LIN {X 0,Y 514.336,Z 499.289,A -85,B 0,C 180,E1 19058.473,E2 19058.473} C_VEL
LIN {X 0,Y 521.666,Z 511.936,A -85,B 0,C 180,E1 19056.114,E2 19056.114} C_VEL
LIN {X 0,Y 522.287,Z 513.297,A -85,B 0,C 180,E1 19055.918,E2 19055.918} C_VEL
LIN {X 0,Y 507.153,Z 734.617,A -85,B 0,C 180,E1 19052.471,E2 19052.471} C_VEL
LIN {X 0,Y 501.246,Z 821.128,A -85,B 0,C 180,E1 19051.105,E2 19051.105} C_VEL
LIN {X 0,Y 497.966,Z 849.233,A -85,B 0,C 180,E1 19050.568,E2 19050.568} C_VEL
LIN {X 0,Y 493.711,Z 874.723,A -85,B 0,C 180,E1 19049.927,E2 19049.927} C_VEL
LIN {X 0,Y 489.478,Z 895.998,A -85,B 0,C 180,E1 19049.256,E2 19049.256} C_VEL
LIN {X 0,Y 484.89,Z 916.021,A -85,B 0,C 180,E1 19048.501,E2 19048.501} C_VEL
LIN {X 0,Y 479.636,Z 936.391,A -85,B 0,C 180,E1 19047.593,E2 19047.593} C_VEL
LIN {X 0,Y 472.466,Z 961.41,A -85,B 0,C 180,E1 19046.272,E2 19046.272} C_VEL
LIN {X 0,Y 464.663,Z 985.247,A -85,B 0,C 180,E1 19044.746,E2 19044.746} C_VEL
LIN {X 0,Y 457.779,Z 1004.83,A -85,B 0,C 180,E1 19043.281,E2 19043.281} C_VEL
LIN {X 0,Y 450.93,Z 1023.119,A -85,B 0,C 180,E1 19041.714,E2 19041.714} C_VEL
LIN {X 0,Y 442.952,Z 1043.356,A -85,B 0,C 180,E1 19039.725,E2 19039.725} C_VEL
LIN {X 0,Y 434.117,Z 1064.457,A -85,B 0,C 180,E1 19037.283,E2 19037.283} C_VEL
LIN {X 0,Y 427.056,Z 1080.83,A -85,B 0,C 180,E1 19035.092,E2 19035.092} C_VEL
LIN {X 0,Y 420.572,Z 1095.666,A -85,B 0,C 180,E1 19032.838,E2 19032.838} C_VEL
LIN {X 0,Y 414.005,Z 1110.651,A -85,B 0,C 180,E1 19030.253,E2 19030.253} C_VEL
LIN {X 0,Y 406.387,Z 1128.256,A -85,B 0,C 180,E1 19026.717,E2 19026.717} C_VEL
LIN {X 0,Y 400.867,Z 1141.384,A -85,B 0,C 180,E1 19023.623,E2 19023.623} C_VEL
LIN {X 0,Y 396.527,Z 1152.254,A -85,B 0,C 180,E1 19020.697,E2 19020.697} C_VEL
LIN {X 0,Y 392.827,Z 1162.333,A -85,B 0,C 180,E1 19017.596,E2 19017.596} C_VEL
LIN {X 0,Y 389.21,Z 1173.396,A -85,B 0,C 180,E1 19013.625,E2 19013.625} C_VEL
LIN {X 0,Y 386.872,Z 1181.783,A -85,B 0,C 180,E1 19009.947,E2 19009.947} C_VEL
LIN {X 0,Y 385.478,Z 1187.928,A -85,B 0,C 180,E1 19006.733,E2 19006.733} C_VEL
LIN {X 0,Y 384.662,Z 1192.751,A -85,B 0,C 180,E1 19003.682,E2 19003.682} C_VEL
LIN {X 0,Y 384.204,Z 1196.587,A -85,B 0,C 180,E1 19000.648,E2 19000.648} C_VEL
LIN {X 0,Y 384.01,Z 1199.46,A -85,B 0,C 180,E1 18997.631,E2 18997.631} C_VEL
LIN {X 0,Y 383.947,Z 1201.384,A -85,B 0,C 180,E1 18994.63,E2 18994.63} C_VEL
LIN {X 0,Y 383.945,Z 1202.344,A -85,B 0,C 180,E1 18991.791,E2 18991.791} C_VEL
LIN {X 0,Y 383.945,Z 1202.461,A -85,B 0,C 180,E1 18988.955,E2 18988.955} C_VEL
LIN {X 0,Y 383.943,Z 1201.632,A -85,B 0,C 180,E1 18985.899,E2 18985.899} C_VEL
LIN {X 0,Y 383.992,Z 1199.811,A -85,B 0,C 180,E1 18982.82,E2 18982.82} C_VEL
LIN {X 0,Y 384.164,Z 1197.081,A -85,B 0,C 180,E1 18979.806,E2 18979.806} C_VEL
LIN {X 0,Y 384.565,Z 1193.388,A -85,B 0,C 180,E1 18976.774,E2 18976.774} C_VEL
LIN {X 0,Y 385.339,Z 1188.712,A -85,B 0,C 180,E1 18973.726,E2 18973.726} C_VEL
LIN {X 0,Y 386.553,Z 1183.024,A -85,B 0,C 180,E1 18970.665,E2 18970.665} C_VEL
LIN {X 0,Y 388.357,Z 1176.207,A -85,B 0,C 180,E1 18967.565,E2 18967.565} C_VEL
LIN {X 0,Y 390.867,Z 1168.055,A -85,B 0,C 180,E1 18964.386,E2 18964.386} C_VEL
LIN {X 0,Y 394.947,Z 1156.625,A -85,B 0,C 180,E1 18960.565,E2 18960.565} C_VEL
LIN {X 0,Y 399.901,Z 1143.712,A -85,B 0,C 180,E1 18956.972,E2 18956.972} C_VEL
LIN {X 0,Y 404.792,Z 1131.925,A -85,B 0,C 180,E1 18954.116,E2 18954.116} C_VEL
LIN {X 0,Y 410.265,Z 1119.184,A -85,B 0,C 180,E1 18951.399,E2 18951.399} C_VEL
LIN {X 0,Y 416.577,Z 1104.778,A -85,B 0,C 180,E1 18948.697,E2 18948.697} C_VEL
LIN {X 0,Y 425.211,Z 1085.008,A -85,B 0,C 180,E1 18945.515,E2 18945.515} C_VEL
LIN {X 0,Y 432.324,Z 1068.503,A -85,B 0,C 180,E1 18943.238,E2 18943.238} C_VEL
LIN {X 0,Y 439.276,Z 1052.004,A -85,B 0,C 180,E1 18941.239,E2 18941.239} C_VEL
LIN {X 0,Y 446.663,Z 1033.856,A -85,B 0,C 180,E1 18939.31,E2 18939.31} C_VEL
LIN {X 0,Y 455.882,Z 1009.897,A -85,B 0,C 180,E1 18937.133,E2 18937.133} C_VEL
LIN {X 0,Y 463.244,Z 989.199,A -85,B 0,C 180,E1 18935.54,E2 18935.54} C_VEL
LIN {X 0,Y 469.526,Z 970.341,A -85,B 0,C 180,E1 18934.285,E2 18934.285} C_VEL
LIN {X 0,Y 475.391,Z 951.136,A -85,B 0,C 180,E1 18933.167,E2 18933.167} C_VEL
LIN {X 0,Y 481.322,Z 929.886,A -85,B 0,C 180,E1 18932.106,E2 18932.106} C_VEL
LIN {X 0,Y 488.036,Z 902.402,A -85,B 0,C 180,E1 18930.975,E2 18930.975} C_VEL
LIN {X 0,Y 492.871,Z 878.77,A -85,B 0,C 180,E1 18930.196,E2 18930.196} C_VEL
LIN {X 0,Y 496.583,Z 857.355,A -85,B 0,C 180,E1 18929.628,E2 18929.628} C_VEL
LIN {X 0,Y 499.707,Z 834.953,A -85,B 0,C 180,E1 18929.153,E2 18929.153} C_VEL
LIN {X 0,Y 502.37,Z 806.226,A -85,B 0,C 180,E1 18928.651,E2 18928.651} C_VEL
LIN {X 0,Y 517.218,Z 584.32,A -85,B 0,C 180,E1 18925.194,E2 18925.194} C_VEL
LIN {X 0,Y 522.155,Z 512.95,A -85,B 0,C 180,E1 18924.072,E2 18924.072} C_VEL
LIN {X 0,Y 515.699,Z 501.805,A -85,B 0,C 180,E1 18922.035,E2 18922.035} C_VEL
LIN {X 0,Y 508.977,Z 490.578,A -85,B 0,C 180,E1 18919.659,E2 18919.659} C_VEL
LIN {X 0,Y 502.568,Z 480.516,A -85,B 0,C 180,E1 18917.065,E2 18917.065} C_VEL
LIN {X 0,Y 498.85,Z 474.804,A -85,B 0,C 180,E1 18915.342,E2 18915.342} C_VEL
LIN {X 0,Y 494.845,Z 469.392,A -85,B 0,C 180,E1 18913.258,E2 18913.258} C_VEL
LIN {X 0,Y 491.244,Z 464.512,A -85,B 0,C 180,E1 18911.03,E2 18911.03} C_VEL
LIN {X 0,Y 488.198,Z 460.623,A -85,B 0,C 180,E1 18908.717,E2 18908.717} C_VEL
LIN {X 0,Y 487.346,Z 459.062,A -85,B 0,C 180,E1 18907.901,E2 18907.901} C_VEL
LIN {X 0,Y 484.26,Z 455.669,A -85,B 0,C 180,E1 18904.144,E2 18904.144} C_VEL
LIN {X 0,Y 483.557,Z 453.202,A -85,B 0,C 180,E1 18902.133,E2 18902.133} C_VEL
LIN {X 0,Y 483.631,Z 453.363,A -85,B 0,C 180,E1 18897.109,E2 18897.109} C_VEL
LIN {X 0,Y 485.036,Z 457.019,A -85,B 0,C 180,E1 18894.084,E2 18894.084} C_VEL
LIN {X 0,Y 487.613,Z 459.507,A -85,B 0,C 180,E1 18891.331,E2 18891.331} C_VEL
LIN {X 0,Y 490.183,Z 463.479,A -85,B 0,C 180,E1 18889.183,E2 18889.183} C_VEL
LIN {X 0,Y 491.887,Z 465.368,A -85,B 0,C 180,E1 18888.033,E2 18888.033} C_VEL
LIN {X 0,Y 495.311,Z 469.926,A -85,B 0,C 180,E1 18885.981,E2 18885.981} C_VEL
LIN {X 0,Y 500.203,Z 476.705,A -85,B 0,C 180,E1 18883.51,E2 18883.51} C_VEL
LIN {X 0,Y 504.513,Z 482.766,A -85,B 0,C 180,E1 18881.632,E2 18881.632} C_VEL
LIN {X 0,Y 509.943,Z 490.429,A -85,B 0,C 180,E1 18879.543,E2 18879.543} C_VEL
LIN {X 0,Y 518.713,Z 503.424,A -85,B 0,C 180,E1 18876.603,E2 18876.603} C_VEL
LIN {X 0,Y 522.118,Z 509.067,A -85,B 0,C 180,E1 18875.558,E2 18875.558} C_VEL
LIN {X 0,Y 507.325,Z 724.277,A -85,B 0,C 180,E1 18872.21,E2 18872.21} C_VEL
LIN {X 0,Y 501.73,Z 805.31,A -85,B 0,C 180,E1 18870.931,E2 18870.931} C_VEL
LIN {X 0,Y 498.508,Z 833.243,A -85,B 0,C 180,E1 18870.382,E2 18870.382} C_VEL
LIN {X 0,Y 494.471,Z 858.277,A -85,B 0,C 180,E1 18869.718,E2 18869.718} C_VEL
LIN {X 0,Y 490.363,Z 879.378,A -85,B 0,C 180,E1 18869.026,E2 18869.026} C_VEL
LIN {X 0,Y 485.757,Z 899.843,A -85,B 0,C 180,E1 18868.222,E2 18868.222} C_VEL
LIN {X 0,Y 480.065,Z 922.038,A -85,B 0,C 180,E1 18867.192,E2 18867.192} C_VEL
LIN {X 0,Y 472.51,Z 947.879,A -85,B 0,C 180,E1 18865.744,E2 18865.744} C_VEL
LIN {X 0,Y 465.938,Z 967.878,A -85,B 0,C 180,E1 18864.419,E2 18864.419} C_VEL
LIN {X 0,Y 459.376,Z 986.337,A -85,B 0,C 180,E1 18863.015,E2 18863.015} C_VEL
LIN {X 0,Y 452.562,Z 1004.295,A -85,B 0,C 180,E1 18861.453,E2 18861.453} C_VEL
LIN {X 0,Y 444.578,Z 1024.231,A -85,B 0,C 180,E1 18859.459,E2 18859.459} C_VEL
LIN {X 0,Y 435.572,Z 1045.248,A -85,B 0,C 180,E1 18856.98,E2 18856.98} C_VEL
LIN {X 0,Y 428.495,Z 1061.153,A -85,B 0,C 180,E1 18854.805,E2 18854.805} C_VEL
LIN {X 0,Y 421.79,Z 1075.935,A -85,B 0,C 180,E1 18852.5,E2 18852.5} C_VEL
LIN {X 0,Y 414.34,Z 1092.31,A -85,B 0,C 180,E1 18849.573,E2 18849.573} C_VEL
LIN {X 0,Y 407.177,Z 1107.877,A -85,B 0,C 180,E1 18846.284,E2 18846.284} C_VEL
LIN {X 0,Y 401.812,Z 1119.823,A -85,B 0,C 180,E1 18843.362,E2 18843.362} C_VEL
LIN {X 0,Y 397.504,Z 1129.916,A -85,B 0,C 180,E1 18840.537,E2 18840.537} C_VEL
LIN {X 0,Y 393.556,Z 1139.762,A -85,B 0,C 180,E1 18837.377,E2 18837.377} C_VEL
LIN {X 0,Y 389.661,Z 1150.554,A -85,B 0,C 180,E1 18833.27,E2 18833.27} C_VEL
LIN {X 0,Y 387.29,Z 1158.095,A -85,B 0,C 180,E1 18829.767,E2 18829.767} C_VEL
LIN {X 0,Y 385.802,Z 1163.853,A -85,B 0,C 180,E1 18826.564,E2 18826.564} C_VEL
LIN {X 0,Y 384.832,Z 1168.546,A -85,B 0,C 180,E1 18823.37,E2 18823.37} C_VEL
LIN {X 0,Y 384.304,Z 1172.209,A -85,B 0,C 180,E1 18820.19,E2 18820.19} C_VEL
LIN {X 0,Y 384.054,Z 1174.876,A -85,B 0,C 180,E1 18817.028,E2 18817.028} C_VEL
LIN {X 0,Y 383.964,Z 1176.634,A -85,B 0,C 180,E1 18813.733,E2 18813.733} C_VEL
LIN {X 0,Y 383.95,Z 1177.409,A -85,B 0,C 180,E1 18810,E2 18810} C_VEL
LIN {X 0,Y 383.964,Z 1176.675,A -85,B 0,C 180,E1 18806.267,E2 18806.267} C_VEL
LIN {X 0,Y 384.048,Z 1174.945,A -85,B 0,C 180,E1 18802.972,E2 18802.972} C_VEL
LIN {X 0,Y 384.075,Z 1174.587,A -85,B 0,C 180,E1 18802.483,E2 18802.483} C_VEL
LIN {X 0,Y 383.137,Z 1173.813,A -85,B 0,C 180,E1 18801.338,E2 18801.338} C_VEL
LIN {X 0,Y 377.082,Z 1171.119,A -85,B 0,C 180,E1 18798.109,E2 18798.109} C_VEL
LIN {X 0,Y 376.701,Z 1170.137,A -85,B 0,C 180,E1 18797.275,E2 18797.275} C_VEL
LIN {X 0,Y 377.746,Z 1165.009,A -85,B 0,C 180,E1 18793.548,E2 18793.548} C_VEL
LIN {X 0,Y 379.241,Z 1159.399,A -85,B 0,C 180,E1 18790.263,E2 18790.263} C_VEL
LIN {X 0,Y 381.436,Z 1152.594,A -85,B 0,C 180,E1 18786.942,E2 18786.942} C_VEL
LIN {X 0,Y 384.593,Z 1144.069,A -85,B 0,C 180,E1 18783.426,E2 18783.426} C_VEL
LIN {X 0,Y 389.595,Z 1131.982,A -85,B 0,C 180,E1 18779.289,E2 18779.289} C_VEL
LIN {X 0,Y 394.485,Z 1120.971,A -85,B 0,C 180,E1 18776.109,E2 18776.109} C_VEL
LIN {X 0,Y 399.733,Z 1109.743,A -85,B 0,C 180,E1 18773.287,E2 18773.287} C_VEL
LIN {X 0,Y 405.907,Z 1096.826,A -85,B 0,C 180,E1 18770.447,E2 18770.447} C_VEL
LIN {X 0,Y 414.365,Z 1079.157,A -85,B 0,C 180,E1 18767.12,E2 18767.12} C_VEL
LIN {X 0,Y 422.034,Z 1062.829,A -85,B 0,C 180,E1 18764.512,E2 18764.512} C_VEL
LIN {X 0,Y 429.08,Z 1047.553,A -85,B 0,C 180,E1 18762.381,E2 18762.381} C_VEL
LIN {X 0,Y 436.644,Z 1030.627,A -85,B 0,C 180,E1 18760.313,E2 18760.313} C_VEL
LIN {X 0,Y 446.241,Z 1007.9,A -85,B 0,C 180,E1 18757.936,E2 18757.936} C_VEL
LIN {X 0,Y 453.74,Z 988.819,A -85,B 0,C 180,E1 18756.244,E2 18756.244} C_VEL
LIN {X 0,Y 460.515,Z 970.415,A -85,B 0,C 180,E1 18754.823,E2 18754.823} C_VEL
LIN {X 0,Y 466.515,Z 952.797,A -85,B 0,C 180,E1 18753.628,E2 18753.628} C_VEL
LIN {X 0,Y 472.745,Z 932.837,A -85,B 0,C 180,E1 18752.447,E2 18752.447} C_VEL
LIN {X 0,Y 479.8,Z 907.755,A -85,B 0,C 180,E1 18751.192,E2 18751.192} C_VEL
LIN {X 0,Y 485.738,Z 882.561,A -85,B 0,C 180,E1 18750.17,E2 18750.17} C_VEL
LIN {X 0,Y 490.062,Z 861.218,A -85,B 0,C 180,E1 18749.456,E2 18749.456} C_VEL
LIN {X 0,Y 493.656,Z 840.065,A -85,B 0,C 180,E1 18748.875,E2 18748.875} C_VEL
LIN {X 0,Y 496.845,Z 816.624,A -85,B 0,C 180,E1 18748.365,E2 18748.365} C_VEL
LIN {X 0,Y 499.925,Z 780.742,A -85,B 0,C 180,E1 18747.765,E2 18747.765} C_VEL
LIN {X 0,Y 515.453,Z 558.007,A -85,B 0,C 180,E1 18744.299,E2 18744.299} C_VEL
LIN {X 0,Y 518.584,Z 513.689,A -85,B 0,C 180,E1 18743.59,E2 18743.59} C_VEL
LIN {X 0,Y 510.496,Z 501.292,A -85,B 0,C 180,E1 18740.914,E2 18740.914} C_VEL
LIN {X 0,Y 503.874,Z 491.617,A -85,B 0,C 180,E1 18738.392,E2 18738.392} C_VEL
LIN {X 0,Y 499.546,Z 485.536,A -85,B 0,C 180,E1 18736.513,E2 18736.513} C_VEL
LIN {X 0,Y 496.88,Z 481.827,A -85,B 0,C 180,E1 18735.225,E2 18735.225} C_VEL
LIN {X 0,Y 493.53,Z 477.194,A -85,B 0,C 180,E1 18733.414,E2 18733.414} C_VEL
LIN {X 0,Y 490.037,Z 472.267,A -85,B 0,C 180,E1 18731.177,E2 18731.177} C_VEL
LIN {X 0,Y 487.021,Z 468.411,A -85,B 0,C 180,E1 18728.798,E2 18728.798} C_VEL
LIN {X 0,Y 486.273,Z 466.929,A -85,B 0,C 180,E1 18728.038,E2 18728.038} C_VEL
LIN {X 0,Y 483.192,Z 463.339,A -85,B 0,C 180,E1 18723.916,E2 18723.916} C_VEL
LIN {X 0,Y 482.689,Z 461.161,A -85,B 0,C 180,E1 18722.018,E2 18722.018} C_VEL
LIN {X 0,Y 482.758,Z 461.298,A -85,B 0,C 180,E1 18718.101,E2 18718.101} C_VEL
LIN {X 0,Y 484.664,Z 465.68,A -85,B 0,C 180,E1 18714.079,E2 18714.079} C_VEL
LIN {X 0,Y 486.62,Z 467.409,A -85,B 0,C 180,E1 18712.038,E2 18712.038} C_VEL
LIN {X 0,Y 489.444,Z 471.765,A -85,B 0,C 180,E1 18709.643,E2 18709.643} C_VEL
LIN {X 0,Y 490.79,Z 473.291,A -85,B 0,C 180,E1 18708.721,E2 18708.721} C_VEL
LIN {X 0,Y 494.745,Z 478.782,A -85,B 0,C 180,E1 18706.322,E2 18706.322} C_VEL
LIN {X 0,Y 498.948,Z 484.683,A -85,B 0,C 180,E1 18704.184,E2 18704.184} C_VEL
LIN {X 0,Y 505.315,Z 494.859,A -85,B 0,C 180,E1 18701.393,E2 18701.393} C_VEL
LIN {X 0,Y 512.231,Z 506.445,A -85,B 0,C 180,E1 18698.801,E2 18698.801} C_VEL
LIN {X 0,Y 518.7,Z 517.874,A -85,B 0,C 180,E1 18696.655,E2 18696.655} C_VEL
LIN {X 0,Y 503.228,Z 738.076,A -85,B 0,C 180,E1 18693.226,E2 18693.226} C_VEL
LIN {X 0,Y 497.396,Z 820.991,A -85,B 0,C 180,E1 18691.915,E2 18691.915} C_VEL
LIN {X 0,Y 494.008,Z 849.281,A -85,B 0,C 180,E1 18691.374,E2 18691.374} C_VEL
LIN {X 0,Y 489.714,Z 874.468,A -85,B 0,C 180,E1 18690.744,E2 18690.744} C_VEL
LIN {X 0,Y 485.383,Z 895.74,A -85,B 0,C 180,E1 18690.079,E2 18690.079} C_VEL
LIN {X 0,Y 480.691,Z 915.761,A -85,B 0,C 180,E1 18689.327,E2 18689.327} C_VEL
LIN {X 0,Y 475.177,Z 936.612,A -85,B 0,C 180,E1 18688.402,E2 18688.402} C_VEL
LIN {X 0,Y 467.654,Z 962.063,A -85,B 0,C 180,E1 18687.053,E2 18687.053} C_VEL
LIN {X 0,Y 459.937,Z 985.028,A -85,B 0,C 180,E1 18685.581,E2 18685.581} C_VEL
LIN {X 0,Y 453.16,Z 1003.821,A -85,B 0,C 180,E1 18684.179,E2 18684.179} C_VEL
LIN {X 0,Y 446.355,Z 1021.501,A -85,B 0,C 180,E1 18682.676,E2 18682.676} C_VEL
LIN {X 0,Y 439.084,Z 1039.394,A -85,B 0,C 180,E1 18680.942,E2 18680.942} C_VEL
LIN {X 0,Y 430.172,Z 1060.455,A -85,B 0,C 180,E1 18678.581,E2 18678.581} C_VEL
LIN {X 0,Y 421.59,Z 1079.621,A -85,B 0,C 180,E1 18676.037,E2 18676.037} C_VEL
LIN {X 0,Y 414.823,Z 1094.533,A -85,B 0,C 180,E1 18673.77,E2 18673.77} C_VEL
LIN {X 0,Y 408.469,Z 1108.461,A -85,B 0,C 180,E1 18671.369,E2 18671.369} C_VEL
LIN {X 0,Y 402.092,Z 1122.506,A -85,B 0,C 180,E1 18668.619,E2 18668.619} C_VEL
LIN {X 0,Y 394.623,Z 1139.351,A -85,B 0,C 180,E1 18664.756,E2 18664.756} C_VEL
LIN {X 0,Y 389.639,Z 1151.167,A -85,B 0,C 180,E1 18661.566,E2 18661.566} C_VEL
LIN {X 0,Y 385.737,Z 1161.118,A -85,B 0,C 180,E1 18658.486,E2 18658.486} C_VEL
LIN {X 0,Y 382.35,Z 1170.7,A -85,B 0,C 180,E1 18655.064,E2 18655.064} C_VEL
LIN {X 0,Y 379.258,Z 1180.887,A -85,B 0,C 180,E1 18650.687,E2 18650.687} C_VEL
LIN {X 0,Y 377.652,Z 1187.396,A -85,B 0,C 180,E1 18647.249,E2 18647.249} C_VEL
LIN {X 0,Y 376.724,Z 1192.483,A -85,B 0,C 180,E1 18643.976,E2 18643.976} C_VEL
LIN {X 0,Y 376.224,Z 1196.321,A -85,B 0,C 180,E1 18640.876,E2 18640.876} C_VEL
LIN {X 0,Y 376.015,Z 1199.196,A -85,B 0,C 180,E1 18637.794,E2 18637.794} C_VEL
LIN {X 0,Y 375.953,Z 1201.05,A -85,B 0,C 180,E1 18634.882,E2 18634.882} C_VEL
LIN {X 0,Y 375.949,Z 1202.081,A -85,B 0,C 180,E1 18631.829,E2 18631.829} C_VEL
LIN {X 0,Y 375.95,Z 1202.198,A -85,B 0,C 180,E1 18628.933,E2 18628.933} C_VEL
LIN {X 0,Y 375.946,Z 1201.387,A -85,B 0,C 180,E1 18625.851,E2 18625.851} C_VEL
LIN {X 0,Y 376.005,Z 1199.547,A -85,B 0,C 180,E1 18622.667,E2 18622.667} C_VEL
LIN {X 0,Y 376.184,Z 1196.789,A -85,B 0,C 180,E1 18619.564,E2 18619.564} C_VEL
LIN {X 0,Y 376.654,Z 1192.906,A -85,B 0,C 180,E1 18616.334,E2 18616.334} C_VEL
LIN {X 0,Y 377.487,Z 1188.179,A -85,B 0,C 180,E1 18613.219,E2 18613.219} C_VEL
LIN {X 0,Y 378.906,Z 1182.17,A -85,B 0,C 180,E1 18609.959,E2 18609.959} C_VEL
LIN {X 0,Y 381.081,Z 1174.564,A -85,B 0,C 180,E1 18606.496,E2 18606.496} C_VEL
LIN {X 0,Y 384.895,Z 1163.457,A -85,B 0,C 180,E1 18602.29,E2 18602.29} C_VEL
LIN {X 0,Y 389.044,Z 1152.603,A -85,B 0,C 180,E1 18598.854,E2 18598.854} C_VEL
LIN {X 0,Y 393.608,Z 1141.677,A -85,B 0,C 180,E1 18595.848,E2 18595.848} C_VEL
LIN {X 0,Y 399.04,Z 1129.249,A -85,B 0,C 180,E1 18592.853,E2 18592.853} C_VEL
LIN {X 0,Y 406.354,Z 1113.12,A -85,B 0,C 180,E1 18589.49,E2 18589.49} C_VEL
LIN {X 0,Y 413.642,Z 1097.059,A -85,B 0,C 180,E1 18586.647,E2 18586.647} C_VEL
LIN {X 0,Y 420.509,Z 1081.911,A -85,B 0,C 180,E1 18584.3,E2 18584.3} C_VEL
LIN {X 0,Y 427.535,Z 1066.17,A -85,B 0,C 180,E1 18582.153,E2 18582.153} C_VEL
LIN {X 0,Y 435.234,Z 1048.451,A -85,B 0,C 180,E1 18580.036,E2 18580.036} C_VEL
LIN {X 0,Y 444.756,Z 1025.434,A -85,B 0,C 180,E1 18577.69,E2 18577.69} C_VEL
LIN {X 0,Y 452.304,Z 1005.911,A -85,B 0,C 180,E1 18575.995,E2 18575.995} C_VEL
LIN {X 0,Y 459.066,Z 987.286,A -85,B 0,C 180,E1 18574.584,E2 18574.584} C_VEL
LIN {X 0,Y 465.827,Z 967.344,A -85,B 0,C 180,E1 18573.277,E2 18573.277} C_VEL
LIN {X 0,Y 473.448,Z 942.736,A -85,B 0,C 180,E1 18571.901,E2 18571.901} C_VEL
LIN {X 0,Y 480.033,Z 918.088,A -85,B 0,C 180,E1 18570.774,E2 18570.774} C_VEL
LIN {X 0,Y 485.038,Z 896.924,A -85,B 0,C 180,E1 18569.968,E2 18569.968} C_VEL
LIN {X 0,Y 489.485,Z 875.199,A -85,B 0,C 180,E1 18569.282,E2 18569.282} C_VEL
LIN {X 0,Y 493.495,Z 851.865,A -85,B 0,C 180,E1 18568.692,E2 18568.692} C_VEL
LIN {X 0,Y 497.217,Z 821.963,A -85,B 0,C 180,E1 18568.108,E2 18568.108} C_VEL
LIN {X 0,Y 501.928,Z 755.768,A -85,B 0,C 180,E1 18567.056,E2 18567.056} C_VEL
LIN {X 0,Y 517.35,Z 534.967,A -85,B 0,C 180,E1 18563.617,E2 18563.617} C_VEL
LIN {X 0,Y 518.578,Z 517.678,A -85,B 0,C 180,E1 18563.343,E2 18563.343} C_VEL
LIN {X 0,Y 511.57,Z 505.471,A -85,B 0,C 180,E1 18561.018,E2 18561.018} C_VEL
LIN {X 0,Y 504.833,Z 494.213,A -85,B 0,C 180,E1 18558.476,E2 18558.476} C_VEL
LIN {X 0,Y 498.44,Z 484.005,A -85,B 0,C 180,E1 18555.653,E2 18555.653} C_VEL
LIN {X 0,Y 493.462,Z 477.084,A -85,B 0,C 180,E1 18553.058,E2 18553.058} C_VEL
LIN {X 0,Y 489.925,Z 472.243,A -85,B 0,C 180,E1 18550.822,E2 18550.822} C_VEL
LIN {X 0,Y 486.957,Z 468.311,A -85,B 0,C 180,E1 18548.502,E2 18548.502} C_VEL
LIN {X 0,Y 486.245,Z 466.949,A -85,B 0,C 180,E1 18547.8,E2 18547.8} C_VEL
LIN {X 0,Y 483.22,Z 463.549,A -85,B 0,C 180,E1 18544.034,E2 18544.034} C_VEL
LIN {X 0,Y 482.543,Z 461.136,A -85,B 0,C 180,E1 18542.019,E2 18542.019} C_VEL
LIN {X 0,Y 482.631,Z 461.368,A -85,B 0,C 180,E1 18537.15,E2 18537.15} C_VEL
LIN {X 0,Y 484.145,Z 465.133,A -85,B 0,C 180,E1 18533.954,E2 18533.954} C_VEL
LIN {X 0,Y 486.446,Z 467.331,A -85,B 0,C 180,E1 18531.489,E2 18531.489} C_VEL
LIN {X 0,Y 489.049,Z 471.365,A -85,B 0,C 180,E1 18529.277,E2 18529.277} C_VEL
LIN {X 0,Y 490.559,Z 473.066,A -85,B 0,C 180,E1 18528.239,E2 18528.239} C_VEL
LIN {X 0,Y 494.723,Z 478.899,A -85,B 0,C 180,E1 18525.725,E2 18525.725} C_VEL
LIN {X 0,Y 498.62,Z 484.252,A -85,B 0,C 180,E1 18523.755,E2 18523.755} C_VEL
LIN {X 0,Y 502.729,Z 490.13,A -85,B 0,C 180,E1 18521.924,E2 18521.924} C_VEL
LIN {X 0,Y 508.137,Z 497.92,A -85,B 0,C 180,E1 18519.797,E2 18519.797} C_VEL
LIN {X 0,Y 516.54,Z 510.577,A -85,B 0,C 180,E1 18516.922,E2 18516.922} C_VEL
LIN {X 0,Y 518.519,Z 513.964,A -85,B 0,C 180,E1 18516.292,E2 18516.292} C_VEL
LIN {X 0,Y 503.283,Z 729.841,A -85,B 0,C 180,E1 18512.933,E2 18512.933} C_VEL
LIN {X 0,Y 497.871,Z 805.809,A -85,B 0,C 180,E1 18511.733,E2 18511.733} C_VEL
LIN {X 0,Y 494.513,Z 834.039,A -85,B 0,C 180,E1 18511.177,E2 18511.177} C_VEL
LIN {X 0,Y 490.451,Z 858.66,A -85,B 0,C 180,E1 18510.524,E2 18510.524} C_VEL
LIN {X 0,Y 486.27,Z 879.653,A -85,B 0,C 180,E1 18509.839,E2 18509.839} C_VEL
LIN {X 0,Y 481.556,Z 900.117,A -85,B 0,C 180,E1 18509.038,E2 18509.038} C_VEL
LIN {X 0,Y 475.787,Z 922.096,A -85,B 0,C 180,E1 18508.022,E2 18508.022} C_VEL
LIN {X 0,Y 467.931,Z 948.312,A -85,B 0,C 180,E1 18506.556,E2 18506.556} C_VEL
LIN {X 0,Y 461.202,Z 968.25,A -85,B 0,C 180,E1 18505.237,E2 18505.237} C_VEL
LIN {X 0,Y 454.498,Z 986.61,A -85,B 0,C 180,E1 18503.839,E2 18503.839} C_VEL
LIN {X 0,Y 447.495,Z 1004.569,A -85,B 0,C 180,E1 18502.275,E2 18502.275} C_VEL
LIN {X 0,Y 439.564,Z 1023.79,A -85,B 0,C 180,E1 18500.351,E2 18500.351} C_VEL
LIN {X 0,Y 430.196,Z 1045.024,A -85,B 0,C 180,E1 18497.852,E2 18497.852} C_VEL
LIN {X 0,Y 422.645,Z 1061.428,A -85,B 0,C 180,E1 18495.598,E2 18495.598} C_VEL
LIN {X 0,Y 415.693,Z 1076.211,A -85,B 0,C 180,E1 18493.275,E2 18493.275} C_VEL
LIN {X 0,Y 407.942,Z 1092.586,A -85,B 0,C 180,E1 18490.32,E2 18490.32} C_VEL
LIN {X 0,Y 400.416,Z 1108.295,A -85,B 0,C 180,E1 18486.957,E2 18486.957} C_VEL
LIN {X 0,Y 394.877,Z 1120.099,A -85,B 0,C 180,E1 18484.027,E2 18484.027} C_VEL
LIN {X 0,Y 390.341,Z 1130.192,A -85,B 0,C 180,E1 18481.159,E2 18481.159} C_VEL
LIN {X 0,Y 386.188,Z 1140.037,A -85,B 0,C 180,E1 18477.944,E2 18477.944} C_VEL
LIN {X 0,Y 382.07,Z 1150.816,A -85,B 0,C 180,E1 18473.766,E2 18473.766} C_VEL
LIN {X 0,Y 379.545,Z 1158.367,A -85,B 0,C 180,E1 18470.188,E2 18470.188} C_VEL
LIN {X 0,Y 377.949,Z 1164.123,A -85,B 0,C 180,E1 18466.918,E2 18466.918} C_VEL
LIN {X 0,Y 376.92,Z 1168.814,A -85,B 0,C 180,E1 18463.656,E2 18463.656} C_VEL
LIN {X 0,Y 376.342,Z 1172.475,A -85,B 0,C 180,E1 18460.408,E2 18460.408} C_VEL
LIN {X 0,Y 376.072,Z 1175.14,A -85,B 0,C 180,E1 18457.178,E2 18457.178} C_VEL
LIN {X 0,Y 375.97,Z 1176.897,A -85,B 0,C 180,E1 18453.812,E2 18453.812} C_VEL
LIN {X 0,Y 375.954,Z 1177.672,A -85,B 0,C 180,E1 18450,E2 18450} C_VEL
LIN {X 0,Y 375.97,Z 1176.938,A -85,B 0,C 180,E1 18446.188,E2 18446.188} C_VEL
LIN {X 0,Y 376.064,Z 1175.208,A -85,B 0,C 180,E1 18442.822,E2 18442.822} C_VEL
LIN {X 0,Y 376.331,Z 1172.57,A -85,B 0,C 180,E1 18439.591,E2 18439.591} C_VEL
LIN {X 0,Y 376.701,Z 1170.137,A -85,B 0,C 180,E1 18437.275,E2 18437.275} C_VEL
LIN {X 0,Y 375.953,Z 1168.761,A -85,B 0,C 180,E1 18436.12,E2 18436.12} C_VEL
LIN {X 0,Y 370.608,Z 1164.818,A -85,B 0,C 180,E1 18432.924,E2 18432.924} C_VEL
LIN {X 0,Y 370.384,Z 1163.436,A -85,B 0,C 180,E1 18431.999,E2 18431.999} C_VEL
LIN {X 0,Y 373.048,Z 1155.068,A -85,B 0,C 180,E1 18427.463,E2 18427.463} C_VEL
LIN {X 0,Y 376.016,Z 1147.133,A -85,B 0,C 180,E1 18423.976,E2 18423.976} C_VEL
LIN {X 0,Y 379.513,Z 1138.773,A -85,B 0,C 180,E1 18420.83,E2 18420.83} C_VEL
LIN {X 0,Y 383.817,Z 1129.234,A -85,B 0,C 180,E1 18417.722,E2 18417.722} C_VEL
LIN {X 0,Y 389.813,Z 1116.753,A -85,B 0,C 180,E1 18414.21,E2 18414.21} C_VEL
LIN {X 0,Y 397.256,Z 1101.581,A -85,B 0,C 180,E1 18410.635,E2 18410.635} C_VEL
LIN {X 0,Y 403.782,Z 1088.477,A -85,B 0,C 180,E1 18407.979,E2 18407.979} C_VEL
LIN {X 0,Y 410.663,Z 1074.59,A -85,B 0,C 180,E1 18405.513,E2 18405.513} C_VEL
LIN {X 0,Y 418.5,Z 1058.535,A -85,B 0,C 180,E1 18403.023,E2 18403.023} C_VEL
LIN {X 0,Y 428.388,Z 1037.47,A -85,B 0,C 180,E1 18400.251,E2 18400.251} C_VEL
LIN {X 0,Y 435.961,Z 1020.477,A -85,B 0,C 180,E1 18398.339,E2 18398.339} C_VEL
LIN {X 0,Y 443.004,Z 1003.86,A -85,B 0,C 180,E1 18396.696,E2 18396.696} C_VEL
LIN {X 0,Y 450.074,Z 986.172,A -85,B 0,C 180,E1 18395.162,E2 18395.162} C_VEL
LIN {X 0,Y 457.591,Z 966.016,A -85,B 0,C 180,E1 18393.644,E2 18393.644} C_VEL
LIN {X 0,Y 466.331,Z 939.98,A -85,B 0,C 180,E1 18391.995,E2 18391.995} C_VEL
LIN {X 0,Y 472.49,Z 919.298,A -85,B 0,C 180,E1 18390.897,E2 18390.897} C_VEL
LIN {X 0,Y 477.877,Z 899.074,A -85,B 0,C 180,E1 18389.979,E2 18389.979} C_VEL
LIN {X 0,Y 482.713,Z 878.399,A -85,B 0,C 180,E1 18389.184,E2 18389.184} C_VEL
LIN {X 0,Y 487.721,Z 853.349,A -85,B 0,C 180,E1 18388.39,E2 18388.39} C_VEL
LIN {X 0,Y 491.928,Z 825.966,A -85,B 0,C 180,E1 18387.728,E2 18387.728} C_VEL
LIN {X 0,Y 494.502,Z 803.09,A -85,B 0,C 180,E1 18387.303,E2 18387.303} C_VEL
LIN {X 0,Y 509.706,Z 592.245,A -85,B 0,C 180,E1 18384.01,E2 18384.01} C_VEL
LIN {X 0,Y 515.062,Z 518.749,A -85,B 0,C 180,E1 18382.846,E2 18382.846} C_VEL
LIN {X 0,Y 507.998,Z 507.822,A -85,B 0,C 180,E1 18380.419,E2 18380.419} C_VEL
LIN {X 0,Y 502.085,Z 498.987,A -85,B 0,C 180,E1 18378.1,E2 18378.1} C_VEL
LIN {X 0,Y 496.253,Z 490.427,A -85,B 0,C 180,E1 18375.424,E2 18375.424} C_VEL
LIN {X 0,Y 492.058,Z 484.78,A -85,B 0,C 180,E1 18373.155,E2 18373.155} C_VEL
LIN {X 0,Y 488.729,Z 480,A -85,B 0,C 180,E1 18370.969,E2 18370.969} C_VEL
LIN {X 0,Y 485.735,Z 475.981,A -85,B 0,C 180,E1 18368.523,E2 18368.523} C_VEL
LIN {X 0,Y 485.054,Z 474.741,A -85,B 0,C 180,E1 18367.82,E2 18367.82} C_VEL
LIN {X 0,Y 482.118,Z 471.08,A -85,B 0,C 180,E1 18363.686,E2 18363.686} C_VEL
LIN {X 0,Y 481.715,Z 469.102,A -85,B 0,C 180,E1 18362.022,E2 18362.022} C_VEL
LIN {X 0,Y 481.77,Z 469.348,A -85,B 0,C 180,E1 18358.097,E2 18358.097} C_VEL
LIN {X 0,Y 483.596,Z 473.562,A -85,B 0,C 180,E1 18354.185,E2 18354.185} C_VEL
LIN {X 0,Y 485.523,Z 475.375,A -85,B 0,C 180,E1 18352.129,E2 18352.129} C_VEL
LIN {X 0,Y 488.31,Z 479.648,A -85,B 0,C 180,E1 18349.738,E2 18349.738} C_VEL
LIN {X 0,Y 489.549,Z 481.131,A -85,B 0,C 180,E1 18348.871,E2 18348.871} C_VEL
LIN {X 0,Y 493.348,Z 486.492,A -85,B 0,C 180,E1 18346.522,E2 18346.522} C_VEL
LIN {X 0,Y 497.487,Z 492.403,A -85,B 0,C 180,E1 18344.376,E2 18344.376} C_VEL
LIN {X 0,Y 503.693,Z 502.587,A -85,B 0,C 180,E1 18341.601,E2 18341.601} C_VEL
LIN {X 0,Y 510.143,Z 513.599,A -85,B 0,C 180,E1 18339.131,E2 18339.131} C_VEL
LIN {X 0,Y 515.186,Z 522.673,A -85,B 0,C 180,E1 18337.399,E2 18337.399} C_VEL
LIN {X 0,Y 499.239,Z 743.742,A -85,B 0,C 180,E1 18333.959,E2 18333.959} C_VEL
LIN {X 0,Y 493.637,Z 820.961,A -85,B 0,C 180,E1 18332.736,E2 18332.736} C_VEL
LIN {X 0,Y 490.134,Z 849.421,A -85,B 0,C 180,E1 18332.192,E2 18332.192} C_VEL
LIN {X 0,Y 485.797,Z 874.321,A -85,B 0,C 180,E1 18331.572,E2 18331.572} C_VEL
LIN {X 0,Y 481.437,Z 895.276,A -85,B 0,C 180,E1 18330.922,E2 18330.922} C_VEL
LIN {X 0,Y 476.593,Z 915.5,A -85,B 0,C 180,E1 18330.168,E2 18330.168} C_VEL
LIN {X 0,Y 470.988,Z 936.219,A -85,B 0,C 180,E1 18329.254,E2 18329.254} C_VEL
LIN {X 0,Y 463.272,Z 961.708,A -85,B 0,C 180,E1 18327.91,E2 18327.91} C_VEL
LIN {X 0,Y 455.417,Z 984.528,A -85,B 0,C 180,E1 18326.453,E2 18326.453} C_VEL
LIN {X 0,Y 448.319,Z 1003.68,A -85,B 0,C 180,E1 18325.027,E2 18325.027} C_VEL
LIN {X 0,Y 441.359,Z 1021.232,A -85,B 0,C 180,E1 18323.535,E2 18323.535} C_VEL
LIN {X 0,Y 433.863,Z 1039.123,A -85,B 0,C 180,E1 18321.799,E2 18321.799} C_VEL
LIN {X 0,Y 424.602,Z 1060.317,A -85,B 0,C 180,E1 18319.413,E2 18319.413} C_VEL
LIN {X 0,Y 415.792,Z 1079.347,A -85,B 0,C 180,E1 18316.872,E2 18316.872} C_VEL
LIN {X 0,Y 408.771,Z 1094.259,A -85,B 0,C 180,E1 18314.588,E2 18314.588} C_VEL
LIN {X 0,Y 402.163,Z 1108.185,A -85,B 0,C 180,E1 18312.165,E2 18312.165} C_VEL
LIN {X 0,Y 395.522,Z 1122.23,A -85,B 0,C 180,E1 18309.384,E2 18309.384} C_VEL
LIN {X 0,Y 387.696,Z 1139.075,A -85,B 0,C 180,E1 18305.469,E2 18305.469} C_VEL
LIN {X 0,Y 382.486,Z 1150.892,A -85,B 0,C 180,E1 18302.227,E2 18302.227} C_VEL
LIN {X 0,Y 378.364,Z 1160.844,A -85,B 0,C 180,E1 18299.093,E2 18299.093} C_VEL
LIN {X 0,Y 374.78,Z 1170.427,A -85,B 0,C 180,E1 18295.607,E2 18295.607} C_VEL
LIN {X 0,Y 371.498,Z 1180.615,A -85,B 0,C 180,E1 18291.14,E2 18291.14} C_VEL
LIN {X 0,Y 369.791,Z 1187.126,A -85,B 0,C 180,E1 18287.628,E2 18287.628} C_VEL
LIN {X 0,Y 368.791,Z 1192.215,A -85,B 0,C 180,E1 18284.283,E2 18284.283} C_VEL
LIN {X 0,Y 368.246,Z 1196.055,A -85,B 0,C 180,E1 18281.115,E2 18281.115} C_VEL
LIN {X 0,Y 368.024,Z 1198.931,A -85,B 0,C 180,E1 18277.964,E2 18277.964} C_VEL
LIN {X 0,Y 367.957,Z 1200.786,A -85,B 0,C 180,E1 18274.988,E2 18274.988} C_VEL
LIN {X 0,Y 367.952,Z 1201.795,A -85,B 0,C 180,E1 18272.024,E2 18272.024} C_VEL
LIN {X 0,Y 367.954,Z 1201.936,A -85,B 0,C 180,E1 18268.91,E2 18268.91} C_VEL
LIN {X 0,Y 367.95,Z 1201.138,A -85,B 0,C 180,E1 18265.792,E2 18265.792} C_VEL
LIN {X 0,Y 368.007,Z 1199.37,A -85,B 0,C 180,E1 18262.624,E2 18262.624} C_VEL
LIN {X 0,Y 368.202,Z 1196.547,A -85,B 0,C 180,E1 18259.359,E2 18259.359} C_VEL
LIN {X 0,Y 368.694,Z 1192.783,A -85,B 0,C 180,E1 18256.142,E2 18256.142} C_VEL
LIN {X 0,Y 369.606,Z 1187.908,A -85,B 0,C 180,E1 18252.85,E2 18252.85} C_VEL
LIN {X 0,Y 371.136,Z 1181.854,A -85,B 0,C 180,E1 18249.499,E2 18249.499} C_VEL
LIN {X 0,Y 373.509,Z 1174.105,A -85,B 0,C 180,E1 18245.905,E2 18245.905} C_VEL
LIN {X 0,Y 377.667,Z 1162.657,A -85,B 0,C 180,E1 18241.521,E2 18241.521} C_VEL
LIN {X 0,Y 382.029,Z 1151.93,A -85,B 0,C 180,E1 18238.084,E2 18238.084} C_VEL
LIN {X 0,Y 386.855,Z 1140.919,A -85,B 0,C 180,E1 18235.019,E2 18235.019} C_VEL
LIN {X 0,Y 392.816,Z 1127.924,A -85,B 0,C 180,E1 18231.864,E2 18231.864} C_VEL
LIN {X 0,Y 401.06,Z 1110.49,A -85,B 0,C 180,E1 18228.269,E2 18228.269} C_VEL
LIN {X 0,Y 407.954,Z 1095.921,A -85,B 0,C 180,E1 18225.693,E2 18225.693} C_VEL
LIN {X 0,Y 415.005,Z 1080.936,A -85,B 0,C 180,E1 18223.367,E2 18223.367} C_VEL
LIN {X 0,Y 422.191,Z 1065.378,A -85,B 0,C 180,E1 18221.243,E2 18221.243} C_VEL
LIN {X 0,Y 430.788,Z 1046.243,A -85,B 0,C 180,E1 18218.965,E2 18218.965} C_VEL
LIN {X 0,Y 440.259,Z 1023.807,A -85,B 0,C 180,E1 18216.709,E2 18216.709} C_VEL
LIN {X 0,Y 447.49,Z 1005.635,A -85,B 0,C 180,E1 18215.137,E2 18215.137} C_VEL
LIN {X 0,Y 454.433,Z 987.01,A -85,B 0,C 180,E1 18213.728,E2 18213.728} C_VEL
LIN {X 0,Y 461.366,Z 967.069,A -85,B 0,C 180,E1 18212.423,E2 18212.423} C_VEL
LIN {X 0,Y 469.232,Z 942.267,A -85,B 0,C 180,E1 18211.043,E2 18211.043} C_VEL
LIN {X 0,Y 475.922,Z 917.813,A -85,B 0,C 180,E1 18209.933,E2 18209.933} C_VEL
LIN {X 0,Y 481.037,Z 896.649,A -85,B 0,C 180,E1 18209.131,E2 18209.131} C_VEL
LIN {X 0,Y 485.499,Z 875.359,A -85,B 0,C 180,E1 18208.463,E2 18208.463} C_VEL
LIN {X 0,Y 489.461,Z 852.884,A -85,B 0,C 180,E1 18207.894,E2 18207.894} C_VEL
LIN {X 0,Y 493.349,Z 823.075,A -85,B 0,C 180,E1 18207.306,E2 18207.306} C_VEL
LIN {X 0,Y 497.411,Z 768.51,A -85,B 0,C 180,E1 18206.434,E2 18206.434} C_VEL
LIN {X 0,Y 513.247,Z 547.156,A -85,B 0,C 180,E1 18202.987,E2 18202.987} C_VEL
LIN {X 0,Y 514.999,Z 522.323,A -85,B 0,C 180,E1 18202.578,E2 18202.578} C_VEL
LIN {X 0,Y 507.085,Z 508.422,A -85,B 0,C 180,E1 18199.796,E2 18199.796} C_VEL
LIN {X 0,Y 500.384,Z 497.216,A -85,B 0,C 180,E1 18197.052,E2 18197.052} C_VEL
LIN {X 0,Y 495.736,Z 489.915,A -85,B 0,C 180,E1 18194.842,E2 18194.842} C_VEL
LIN {X 0,Y 491.885,Z 484.553,A -85,B 0,C 180,E1 18192.742,E2 18192.742} C_VEL
LIN {X 0,Y 488.612,Z 479.971,A -85,B 0,C 180,E1 18190.613,E2 18190.613} C_VEL
LIN {X 0,Y 485.663,Z 475.875,A -85,B 0,C 180,E1 18188.227,E2 18188.227} C_VEL
LIN {X 0,Y 485.019,Z 474.758,A -85,B 0,C 180,E1 18187.582,E2 18187.582} C_VEL
LIN {X 0,Y 482.127,Z 471.278,A -85,B 0,C 180,E1 18183.805,E2 18183.805} C_VEL
LIN {X 0,Y 481.531,Z 469.068,A -85,B 0,C 180,E1 18181.904,E2 18181.904} C_VEL
LIN {X 0,Y 481.619,Z 469.26,A -85,B 0,C 180,E1 18177.263,E2 18177.263} C_VEL
LIN {X 0,Y 483.169,Z 473.126,A -85,B 0,C 180,E1 18173.942,E2 18173.942} C_VEL
LIN {X 0,Y 485.283,Z 475.153,A -85,B 0,C 180,E1 18171.648,E2 18171.648} C_VEL
LIN {X 0,Y 487.917,Z 479.251,A -85,B 0,C 180,E1 18169.372,E2 18169.372} C_VEL
LIN {X 0,Y 489.318,Z 480.915,A -85,B 0,C 180,E1 18168.388,E2 18168.388} C_VEL
LIN {X 0,Y 493.324,Z 486.607,A -85,B 0,C 180,E1 18165.923,E2 18165.923} C_VEL
LIN {X 0,Y 497.161,Z 491.978,A -85,B 0,C 180,E1 18163.946,E2 18163.946} C_VEL
LIN {X 0,Y 502.813,Z 500.046,A -85,B 0,C 180,E1 18161.447,E2 18161.447} C_VEL
LIN {X 0,Y 509.506,Z 510.276,A -85,B 0,C 180,E1 18158.893,E2 18158.893} C_VEL
LIN {X 0,Y 515.01,Z 518.766,A -85,B 0,C 180,E1 18157.038,E2 18157.038} C_VEL
LIN {X 0,Y 499.527,Z 732.467,A -85,B 0,C 180,E1 18153.714,E2 18153.714} C_VEL
LIN {X 0,Y 494.12,Z 806.202,A -85,B 0,C 180,E1 18152.549,E2 18152.549} C_VEL
LIN {X 0,Y 490.657,Z 834.576,A -85,B 0,C 180,E1 18151.991,E2 18151.991} C_VEL
LIN {X 0,Y 486.529,Z 859.043,A -85,B 0,C 180,E1 18151.344,E2 18151.344} C_VEL
LIN {X 0,Y 482.277,Z 879.927,A -85,B 0,C 180,E1 18150.666,E2 18150.666} C_VEL
LIN {X 0,Y 477.456,Z 900.39,A -85,B 0,C 180,E1 18149.869,E2 18149.869} C_VEL
LIN {X 0,Y 471.43,Z 922.815,A -85,B 0,C 180,E1 18148.834,E2 18148.834} C_VEL
LIN {X 0,Y 463.466,Z 948.693,A -85,B 0,C 180,E1 18147.387,E2 18147.387} C_VEL
LIN {X 0,Y 456.633,Z 968.425,A -85,B 0,C 180,E1 18146.085,E2 18146.085} C_VEL
LIN {X 0,Y 449.719,Z 986.884,A -85,B 0,C 180,E1 18144.681,E2 18144.681} C_VEL
LIN {X 0,Y 442.524,Z 1004.842,A -85,B 0,C 180,E1 18143.115,E2 18143.115} C_VEL
LIN {X 0,Y 434.357,Z 1024.064,A -85,B 0,C 180,E1 18141.187,E2 18141.187} C_VEL
LIN {X 0,Y 424.691,Z 1045.3,A -85,B 0,C 180,E1 18138.679,E2 18138.679} C_VEL
LIN {X 0,Y 416.884,Z 1061.704,A -85,B 0,C 180,E1 18136.412,E2 18136.412} C_VEL
LIN {X 0,Y 409.68,Z 1076.487,A -85,B 0,C 180,E1 18134.072,E2 18134.072} C_VEL
LIN {X 0,Y 401.976,Z 1092.106,A -85,B 0,C 180,E1 18131.235,E2 18131.235} C_VEL
LIN {X 0,Y 393.848,Z 1108.43,A -85,B 0,C 180,E1 18127.721,E2 18127.721} C_VEL
LIN {X 0,Y 387.999,Z 1120.375,A -85,B 0,C 180,E1 18124.716,E2 18124.716} C_VEL
LIN {X 0,Y 383.001,Z 1130.97,A -85,B 0,C 180,E1 18121.65,E2 18121.65} C_VEL
LIN {X 0,Y 378.133,Z 1142.102,A -85,B 0,C 180,E1 18117.906,E2 18117.906} C_VEL
LIN {X 0,Y 374.1,Z 1152.119,A -85,B 0,C 180,E1 18113.802,E2 18113.802} C_VEL
LIN {X 0,Y 371.722,Z 1158.932,A -85,B 0,C 180,E1 18110.467,E2 18110.467} C_VEL
LIN {X 0,Y 370.047,Z 1164.639,A -85,B 0,C 180,E1 18107.128,E2 18107.128} C_VEL
LIN {X 0,Y 368.971,Z 1169.281,A -85,B 0,C 180,E1 18103.796,E2 18103.796} C_VEL
LIN {X 0,Y 368.363,Z 1172.896,A -85,B 0,C 180,E1 18100.478,E2 18100.478} C_VEL
LIN {X 0,Y 368.07,Z 1175.624,A -85,B 0,C 180,E1 18097.021,E2 18097.021} C_VEL
LIN {X 0,Y 367.966,Z 1177.521,A -85,B 0,C 180,E1 18092.959,E2 18092.959} C_VEL
LIN {X 0,Y 367.952,Z 1177.815,A -85,B 0,C 180,E1 18089.066,E2 18089.066} C_VEL
LIN {X 0,Y 367.981,Z 1177.044,A -85,B 0,C 180,E1 18085.735,E2 18085.735} C_VEL
LIN {X 0,Y 368.091,Z 1175.362,A -85,B 0,C 180,E1 18082.508,E2 18082.508} C_VEL
LIN {X 0,Y 368.38,Z 1172.762,A -85,B 0,C 180,E1 18079.289,E2 18079.289} C_VEL
LIN {X 0,Y 368.997,Z 1169.2,A -85,B 0,C 180,E1 18076.045,E2 18076.045} C_VEL
LIN {X 0,Y 370.073,Z 1164.538,A -85,B 0,C 180,E1 18072.711,E2 18072.711} C_VEL
LIN {X 0,Y 370.384,Z 1163.436,A -85,B 0,C 180,E1 18071.999,E2 18071.999} C_VEL
LIN {X 0,Y 369.982,Z 1161.673,A -85,B 0,C 180,E1 18070.831,E2 18070.831} C_VEL
LIN {X 0,Y 365.61,Z 1156.567,A -85,B 0,C 180,E1 18067.596,E2 18067.596} C_VEL
LIN {X 0,Y 365.652,Z 1154.727,A -85,B 0,C 180,E1 18066.679,E2 18066.679} C_VEL
LIN {X 0,Y 368.741,Z 1147.009,A -85,B 0,C 180,E1 18063.249,E2 18063.249} C_VEL
LIN {X 0,Y 372.468,Z 1138.597,A -85,B 0,C 180,E1 18060.046,E2 18060.046} C_VEL
LIN {X 0,Y 377.308,Z 1128.499,A -85,B 0,C 180,E1 18056.733,E2 18056.733} C_VEL
LIN {X 0,Y 384.273,Z 1114.645,A -85,B 0,C 180,E1 18052.868,E2 18052.868} C_VEL
LIN {X 0,Y 391.202,Z 1101.164,A -85,B 0,C 180,E1 18049.712,E2 18049.712} C_VEL
LIN {X 0,Y 397.895,Z 1088.242,A -85,B 0,C 180,E1 18047.079,E2 18047.079} C_VEL
LIN {X 0,Y 404.857,Z 1074.705,A -85,B 0,C 180,E1 18044.663,E2 18044.663} C_VEL
LIN {X 0,Y 412.89,Z 1058.803,A -85,B 0,C 180,E1 18042.183,E2 18042.183} C_VEL
LIN {X 0,Y 423.091,Z 1037.738,A -85,B 0,C 180,E1 18039.397,E2 18039.397} C_VEL
LIN {X 0,Y 430.901,Z 1020.743,A -85,B 0,C 180,E1 18037.48,E2 18037.48} C_VEL
LIN {X 0,Y 438.289,Z 1003.805,A -85,B 0,C 180,E1 18035.807,E2 18035.807} C_VEL
LIN {X 0,Y 445.778,Z 985.533,A -85,B 0,C 180,E1 18034.229,E2 18034.229} C_VEL
LIN {X 0,Y 454.346,Z 963.059,A -85,B 0,C 180,E1 18032.558,E2 18032.558} C_VEL
LIN {X 0,Y 462.359,Z 939.342,A -85,B 0,C 180,E1 18031.091,E2 18031.091} C_VEL
LIN {X 0,Y 468.389,Z 919.556,A -85,B 0,C 180,E1 18030.048,E2 18030.048} C_VEL
LIN {X 0,Y 473.897,Z 899.33,A -85,B 0,C 180,E1 18029.134,E2 18029.134} C_VEL
LIN {X 0,Y 478.841,Z 878.653,A -85,B 0,C 180,E1 18028.343,E2 18028.343} C_VEL
LIN {X 0,Y 483.933,Z 853.709,A -85,B 0,C 180,E1 18027.557,E2 18027.557} C_VEL
LIN {X 0,Y 488.234,Z 826.341,A -85,B 0,C 180,E1 18026.899,E2 18026.899} C_VEL
LIN {X 0,Y 490.872,Z 803.409,A -85,B 0,C 180,E1 18026.474,E2 18026.474} C_VEL
LIN {X 0,Y 506.479,Z 592.735,A -85,B 0,C 180,E1 18023.186,E2 18023.186} C_VEL
LIN {X 0,Y 511.663,Z 523.827,A -85,B 0,C 180,E1 18022.104,E2 18022.104} C_VEL
LIN {X 0,Y 503.515,Z 511.116,A -85,B 0,C 180,E1 18019.127,E2 18019.127} C_VEL
LIN {X 0,Y 497.216,Z 501.762,A -85,B 0,C 180,E1 18016.412,E2 18016.412} C_VEL
LIN {X 0,Y 493.705,Z 496.796,A -85,B 0,C 180,E1 18014.665,E2 18014.665} C_VEL
LIN {X 0,Y 490.693,Z 492.474,A -85,B 0,C 180,E1 18012.953,E2 18012.953} C_VEL
LIN {X 0,Y 487.427,Z 487.731,A -85,B 0,C 180,E1 18010.759,E2 18010.759} C_VEL
LIN {X 0,Y 484.515,Z 483.671,A -85,B 0,C 180,E1 18008.306,E2 18008.306} C_VEL
LIN {X 0,Y 483.843,Z 482.553,A -85,B 0,C 180,E1 18007.6,E2 18007.6} C_VEL
LIN {X 0,Y 481.015,Z 478.672,A -85,B 0,C 180,E1 18003.337,E2 18003.337} C_VEL
LIN {X 0,Y 480.71,Z 477.039,A -85,B 0,C 180,E1 18001.907,E2 18001.907} C_VEL
LIN {X 0,Y 480.767,Z 477.231,A -85,B 0,C 180,E1 17998.212,E2 17998.212} C_VEL
LIN {X 0,Y 482.622,Z 481.535,A -85,B 0,C 180,E1 17994.173,E2 17994.173} C_VEL
LIN {X 0,Y 484.364,Z 483.187,A -85,B 0,C 180,E1 17992.289,E2 17992.289} C_VEL
LIN {X 0,Y 487.176,Z 487.531,A -85,B 0,C 180,E1 17989.834,E2 17989.834} C_VEL
LIN {X 0,Y 488.392,Z 489.11,A -85,B 0,C 180,E1 17988.964,E2 17988.964} C_VEL
LIN {X 0,Y 491.958,Z 494.199,A -85,B 0,C 180,E1 17986.722,E2 17986.722} C_VEL
LIN {X 0,Y 496.031,Z 500.12,A -85,B 0,C 180,E1 17984.569,E2 17984.569} C_VEL
LIN {X 0,Y 502.144,Z 510.426,A -85,B 0,C 180,E1 17981.782,E2 17981.782} C_VEL
LIN {X 0,Y 508.145,Z 520.89,A -85,B 0,C 180,E1 17979.437,E2 17979.437} C_VEL
LIN {X 0,Y 511.749,Z 527.564,A -85,B 0,C 180,E1 17978.152,E2 17978.152} C_VEL
LIN {X 0,Y 495.447,Z 747.802,A -85,B 0,C 180,E1 17974.728,E2 17974.728} C_VEL
LIN {X 0,Y 489.981,Z 820.932,A -85,B 0,C 180,E1 17973.569,E2 17973.569} C_VEL
LIN {X 0,Y 486.317,Z 849.823,A -85,B 0,C 180,E1 17973.016,E2 17973.016} C_VEL
LIN {X 0,Y 481.983,Z 874.175,A -85,B 0,C 180,E1 17972.414,E2 17972.414} C_VEL
LIN {X 0,Y 477.379,Z 895.768,A -85,B 0,C 180,E1 17971.747,E2 17971.747} C_VEL
LIN {X 0,Y 472.267,Z 916.533,A -85,B 0,C 180,E1 17970.971,E2 17970.971} C_VEL
LIN {X 0,Y 465.995,Z 939.018,A -85,B 0,C 180,E1 17969.97,E2 17969.97} C_VEL
LIN {X 0,Y 457.704,Z 965.04,A -85,B 0,C 180,E1 17968.561,E2 17968.561} C_VEL
LIN {X 0,Y 450.539,Z 985.268,A -85,B 0,C 180,E1 17967.256,E2 17967.256} C_VEL
LIN {X 0,Y 443.382,Z 1004.028,A -85,B 0,C 180,E1 17965.854,E2 17965.854} C_VEL
LIN {X 0,Y 436.184,Z 1021.637,A -85,B 0,C 180,E1 17964.352,E2 17964.352} C_VEL
LIN {X 0,Y 427.693,Z 1041.313,A -85,B 0,C 180,E1 17962.421,E2 17962.421} C_VEL
LIN {X 0,Y 417.868,Z 1062.776,A -85,B 0,C 180,E1 17959.933,E2 17959.933} C_VEL
LIN {X 0,Y 409.851,Z 1079.543,A -85,B 0,C 180,E1 17957.662,E2 17957.662} C_VEL
LIN {X 0,Y 402.498,Z 1094.602,A -85,B 0,C 180,E1 17955.329,E2 17955.329} C_VEL
LIN {X 0,Y 395.552,Z 1108.693,A -85,B 0,C 180,E1 17952.841,E2 17952.841} C_VEL
LIN {X 0,Y 387.562,Z 1125.048,A -85,B 0,C 180,E1 17949.519,E2 17949.519} C_VEL
LIN {X 0,Y 380.275,Z 1139.97,A -85,B 0,C 180,E1 17945.897,E2 17945.897} C_VEL
LIN {X 0,Y 375.14,Z 1151.143,A -85,B 0,C 180,E1 17942.755,E2 17942.755} C_VEL
LIN {X 0,Y 370.648,Z 1161.509,A -85,B 0,C 180,E1 17939.404,E2 17939.404} C_VEL
LIN {X 0,Y 366.386,Z 1172.576,A -85,B 0,C 180,E1 17935.196,E2 17935.196} C_VEL
LIN {X 0,Y 363.465,Z 1181.28,A -85,B 0,C 180,E1 17931.123,E2 17931.123} C_VEL
LIN {X 0,Y 361.806,Z 1187.381,A -85,B 0,C 180,E1 17927.697,E2 17927.697} C_VEL
LIN {X 0,Y 360.823,Z 1192.16,A -85,B 0,C 180,E1 17924.442,E2 17924.442} C_VEL
LIN {X 0,Y 360.254,Z 1195.954,A -85,B 0,C 180,E1 17921.203,E2 17921.203} C_VEL
LIN {X 0,Y 360.026,Z 1198.785,A -85,B 0,C 180,E1 17917.982,E2 17917.982} C_VEL
LIN {X 0,Y 359.959,Z 1200.594,A -85,B 0,C 180,E1 17914.94,E2 17914.94} C_VEL
LIN {X 0,Y 359.957,Z 1201.556,A -85,B 0,C 180,E1 17911.91,E2 17911.91} C_VEL
LIN {X 0,Y 359.959,Z 1201.673,A -85,B 0,C 180,E1 17908.886,E2 17908.886} C_VEL
LIN {X 0,Y 359.953,Z 1200.875,A -85,B 0,C 180,E1 17905.699,E2 17905.699} C_VEL
LIN {X 0,Y 360.012,Z 1199.135,A -85,B 0,C 180,E1 17902.5,E2 17902.5} C_VEL
LIN {X 0,Y 360.222,Z 1196.28,A -85,B 0,C 180,E1 17899.12,E2 17899.12} C_VEL
LIN {X 0,Y 360.785,Z 1192.369,A -85,B 0,C 180,E1 17895.721,E2 17895.721} C_VEL
LIN {X 0,Y 361.74,Z 1187.637,A -85,B 0,C 180,E1 17892.466,E2 17892.466} C_VEL
LIN {X 0,Y 363.37,Z 1181.581,A -85,B 0,C 180,E1 17889.04,E2 17889.04} C_VEL
LIN {X 0,Y 365.838,Z 1174.015,A -85,B 0,C 180,E1 17885.454,E2 17885.454} C_VEL
LIN {X 0,Y 370.271,Z 1162.432,A -85,B 0,C 180,E1 17880.918,E2 17880.918} C_VEL
LIN {X 0,Y 374.903,Z 1151.652,A -85,B 0,C 180,E1 17877.403,E2 17877.403} C_VEL
LIN {X 0,Y 379.724,Z 1141.118,A -85,B 0,C 180,E1 17874.415,E2 17874.415} C_VEL
LIN {X 0,Y 385.675,Z 1128.689,A -85,B 0,C 180,E1 17871.333,E2 17871.333} C_VEL
LIN {X 0,Y 393.759,Z 1112.377,A -85,B 0,C 180,E1 17867.859,E2 17867.859} C_VEL
LIN {X 0,Y 401.957,Z 1095.641,A -85,B 0,C 180,E1 17864.852,E2 17864.852} C_VEL
LIN {X 0,Y 409.162,Z 1080.883,A -85,B 0,C 180,E1 17862.543,E2 17862.543} C_VEL
LIN {X 0,Y 416.462,Z 1065.613,A -85,B 0,C 180,E1 17860.442,E2 17860.442} C_VEL
LIN {X 0,Y 424.528,Z 1048.214,A -85,B 0,C 180,E1 17858.345,E2 17858.345} C_VEL
LIN {X 0,Y 434.782,Z 1024.88,A -85,B 0,C 180,E1 17855.955,E2 17855.955} C_VEL
LIN {X 0,Y 442.778,Z 1005.359,A -85,B 0,C 180,E1 17854.261,E2 17854.261} C_VEL
LIN {X 0,Y 449.909,Z 986.735,A -85,B 0,C 180,E1 17852.855,E2 17852.855} C_VEL
LIN {X 0,Y 457.012,Z 966.793,A -85,B 0,C 180,E1 17851.553,E2 17851.553} C_VEL
LIN {X 0,Y 465.013,Z 942.187,A -85,B 0,C 180,E1 17850.19,E2 17850.19} C_VEL
LIN {X 0,Y 471.915,Z 917.539,A -85,B 0,C 180,E1 17849.077,E2 17849.077} C_VEL
LIN {X 0,Y 477.131,Z 896.426,A -85,B 0,C 180,E1 17848.283,E2 17848.283} C_VEL
LIN {X 0,Y 481.679,Z 875.192,A -85,B 0,C 180,E1 17847.622,E2 17847.622} C_VEL
LIN {X 0,Y 485.687,Z 852.935,A -85,B 0,C 180,E1 17847.061,E2 17847.061} C_VEL
LIN {X 0,Y 489.618,Z 823.757,A -85,B 0,C 180,E1 17846.485,E2 17846.485} C_VEL
LIN {X 0,Y 493.513,Z 773.316,A -85,B 0,C 180,E1 17845.677,E2 17845.677} C_VEL
LIN {X 0,Y 509.74,Z 552.279,A -85,B 0,C 180,E1 17842.237,E2 17842.237} C_VEL
LIN {X 0,Y 511.582,Z 527.175,A -85,B 0,C 180,E1 17841.83,E2 17841.83} C_VEL
LIN {X 0,Y 504.231,Z 514.141,A -85,B 0,C 180,E1 17839.129,E2 17839.129} C_VEL
LIN {X 0,Y 498.325,Z 504.115,A -85,B 0,C 180,E1 17836.614,E2 17836.614} C_VEL
LIN {X 0,Y 494.193,Z 497.469,A -85,B 0,C 180,E1 17834.59,E2 17834.59} C_VEL
LIN {X 0,Y 490.518,Z 492.243,A -85,B 0,C 180,E1 17832.538,E2 17832.538} C_VEL
LIN {X 0,Y 487.473,Z 487.851,A -85,B 0,C 180,E1 17830.519,E2 17830.519} C_VEL
LIN {X 0,Y 484.495,Z 483.686,A -85,B 0,C 180,E1 17828.067,E2 17828.067} C_VEL
LIN {X 0,Y 483.8,Z 482.562,A -85,B 0,C 180,E1 17827.362,E2 17827.362} C_VEL
LIN {X 0,Y 481.092,Z 479.158,A -85,B 0,C 180,E1 17823.694,E2 17823.694} C_VEL
LIN {X 0,Y 480.521,Z 477,A -85,B 0,C 180,E1 17821.789,E2 17821.789} C_VEL
LIN {X 0,Y 480.608,Z 477.151,A -85,B 0,C 180,E1 17817.377,E2 17817.377} C_VEL
LIN {X 0,Y 482.107,Z 481.005,A -85,B 0,C 180,E1 17814.048,E2 17814.048} C_VEL
LIN {X 0,Y 484.177,Z 483.102,A -85,B 0,C 180,E1 17811.748,E2 17811.748} C_VEL
LIN {X 0,Y 486.945,Z 487.3,A -85,B 0,C 180,E1 17809.35,E2 17809.35} C_VEL
LIN {X 0,Y 488.081,Z 488.76,A -85,B 0,C 180,E1 17808.538,E2 17808.538} C_VEL
LIN {X 0,Y 491.931,Z 494.313,A -85,B 0,C 180,E1 17806.123,E2 17806.123} C_VEL
LIN {X 0,Y 495.708,Z 499.702,A -85,B 0,C 180,E1 17804.138,E2 17804.138} C_VEL
LIN {X 0,Y 501.085,Z 507.521,A -85,B 0,C 180,E1 17801.712,E2 17801.712} C_VEL
LIN {X 0,Y 507.524,Z 517.537,A -85,B 0,C 180,E1 17799.199,E2 17799.199} C_VEL
LIN {X 0,Y 511.558,Z 524.04,A -85,B 0,C 180,E1 17797.786,E2 17797.786} C_VEL
LIN {X 0,Y 495.485,Z 740.366,A -85,B 0,C 180,E1 17794.424,E2 17794.424} C_VEL
LIN {X 0,Y 490.452,Z 806.808,A -85,B 0,C 180,E1 17793.373,E2 17793.373} C_VEL
LIN {X 0,Y 486.794,Z 835.762,A -85,B 0,C 180,E1 17792.801,E2 17792.801} C_VEL
LIN {X 0,Y 482.689,Z 859.534,A -85,B 0,C 180,E1 17792.174,E2 17792.174} C_VEL
LIN {X 0,Y 478.221,Z 880.937,A -85,B 0,C 180,E1 17791.48,E2 17791.48} C_VEL
LIN {X 0,Y 473.101,Z 902.068,A -85,B 0,C 180,E1 17790.654,E2 17790.654} C_VEL
LIN {X 0,Y 466.034,Z 927.508,A -85,B 0,C 180,E1 17789.462,E2 17789.462} C_VEL
LIN {X 0,Y 458.463,Z 950.906,A -85,B 0,C 180,E1 17788.12,E2 17788.12} C_VEL
LIN {X 0,Y 451.658,Z 969.972,A -85,B 0,C 180,E1 17786.851,E2 17786.851} C_VEL
LIN {X 0,Y 444.461,Z 988.612,A -85,B 0,C 180,E1 17785.421,E2 17785.421} C_VEL
LIN {X 0,Y 436.262,Z 1008.419,A -85,B 0,C 180,E1 17783.667,E2 17783.667} C_VEL
LIN {X 0,Y 426.086,Z 1031.149,A -85,B 0,C 180,E1 17781.283,E2 17781.283} C_VEL
LIN {X 0,Y 418.047,Z 1048.074,A -85,B 0,C 180,E1 17779.199,E2 17779.199} C_VEL
LIN {X 0,Y 410.297,Z 1063.804,A -85,B 0,C 180,E1 17776.976,E2 17776.976} C_VEL
LIN {X 0,Y 401.675,Z 1080.921,A -85,B 0,C 180,E1 17774.185,E2 17774.185} C_VEL
LIN {X 0,Y 392.894,Z 1097.849,A -85,B 0,C 180,E1 17770.9,E2 17770.9} C_VEL
LIN {X 0,Y 386.604,Z 1110.002,A -85,B 0,C 180,E1 17768.163,E2 17768.163} C_VEL
LIN {X 0,Y 380.881,Z 1121.232,A -85,B 0,C 180,E1 17765.27,E2 17765.27} C_VEL
LIN {X 0,Y 375.692,Z 1131.749,A -85,B 0,C 180,E1 17762.159,E2 17762.159} C_VEL
LIN {X 0,Y 370.43,Z 1143.236,A -85,B 0,C 180,E1 17758.187,E2 17758.187} C_VEL
LIN {X 0,Y 366.398,Z 1152.735,A -85,B 0,C 180,E1 17754.163,E2 17754.163} C_VEL
LIN {X 0,Y 363.908,Z 1159.498,A -85,B 0,C 180,E1 17750.759,E2 17750.759} C_VEL
LIN {X 0,Y 362.15,Z 1165.156,A -85,B 0,C 180,E1 17747.348,E2 17747.348} C_VEL
LIN {X 0,Y 361.024,Z 1169.749,A -85,B 0,C 180,E1 17743.942,E2 17743.942} C_VEL
LIN {X 0,Y 360.344,Z 1173.625,A -85,B 0,C 180,E1 17740.229,E2 17740.229} C_VEL
LIN {X 0,Y 360.041,Z 1176.574,A -85,B 0,C 180,E1 17736.058,E2 17736.058} C_VEL
LIN {X 0,Y 359.962,Z 1177.89,A -85,B 0,C 180,E1 17732.229,E2 17732.229} C_VEL
LIN {X 0,Y 359.959,Z 1178.055,A -85,B 0,C 180,E1 17728.886,E2 17728.886} C_VEL
LIN {X 0,Y 359.987,Z 1177.323,A -85,B 0,C 180,E1 17725.677,E2 17725.677} C_VEL
LIN {X 0,Y 360.106,Z 1175.626,A -85,B 0,C 180,E1 17722.341,E2 17722.341} C_VEL
LIN {X 0,Y 360.414,Z 1173.1,A -85,B 0,C 180,E1 17719.126,E2 17719.126} C_VEL
LIN {X 0,Y 361.093,Z 1169.467,A -85,B 0,C 180,E1 17715.733,E2 17715.733} C_VEL
LIN {X 0,Y 362.247,Z 1164.807,A -85,B 0,C 180,E1 17712.325,E2 17712.325} C_VEL
LIN {X 0,Y 364.06,Z 1159.081,A -85,B 0,C 180,E1 17708.913,E2 17708.913} C_VEL
LIN {X 0,Y 365.652,Z 1154.727,A -85,B 0,C 180,E1 17706.679,E2 17706.679} C_VEL
LIN {X 0,Y 365.604,Z 1152.449,A -85,B 0,C 180,E1 17705.518,E2 17705.518} C_VEL
LIN {X 0,Y 362.428,Z 1146.4,A -85,B 0,C 180,E1 17702.348,E2 17702.348} C_VEL
LIN {X 0,Y 362.814,Z 1144.143,A -85,B 0,C 180,E1 17701.355,E2 17701.355} C_VEL
LIN {X 0,Y 368.541,Z 1132.294,A -85,B 0,C 180,E1 17697.139,E2 17697.139} C_VEL
LIN {X 0,Y 373.981,Z 1121.786,A -85,B 0,C 180,E1 17693.972,E2 17693.972} C_VEL
LIN {X 0,Y 379.947,Z 1110.558,A -85,B 0,C 180,E1 17691.028,E2 17691.028} C_VEL
LIN {X 0,Y 386.876,Z 1097.728,A -85,B 0,C 180,E1 17688.103,E2 17688.103} C_VEL
LIN {X 0,Y 396.429,Z 1079.968,A -85,B 0,C 180,E1 17684.663,E2 17684.663} C_VEL
LIN {X 0,Y 404.498,Z 1064.549,A -85,B 0,C 180,E1 17682.136,E2 17682.136} C_VEL
LIN {X 0,Y 412.472,Z 1048.903,A -85,B 0,C 180,E1 17679.906,E2 17679.906} C_VEL
LIN {X 0,Y 420.722,Z 1032.088,A -85,B 0,C 180,E1 17677.819,E2 17677.819} C_VEL
LIN {X 0,Y 430.684,Z 1010.677,A -85,B 0,C 180,E1 17675.541,E2 17675.541} C_VEL
LIN {X 0,Y 439.665,Z 989.61,A -85,B 0,C 180,E1 17673.661,E2 17673.661} C_VEL
LIN {X 0,Y 446.916,Z 971.366,A -85,B 0,C 180,E1 17672.256,E2 17672.256} C_VEL
LIN {X 0,Y 453.46,Z 953.595,A -85,B 0,C 180,E1 17671.063,E2 17671.063} C_VEL
LIN {X 0,Y 460.155,Z 933.615,A -85,B 0,C 180,E1 17669.891,E2 17669.891} C_VEL
LIN {X 0,Y 467.713,Z 908.525,A -85,B 0,C 180,E1 17668.652,E2 17668.652} C_VEL
LIN {X 0,Y 474.056,Z 883.324,A -85,B 0,C 180,E1 17667.645,E2 17667.645} C_VEL
LIN {X 0,Y 478.652,Z 862.082,A -85,B 0,C 180,E1 17666.947,E2 17666.947} C_VEL
LIN {X 0,Y 482.452,Z 841.073,A -85,B 0,C 180,E1 17666.379,E2 17666.379} C_VEL
LIN {X 0,Y 485.829,Z 817.812,A -85,B 0,C 180,E1 17665.88,E2 17665.88} C_VEL
LIN {X 0,Y 489.148,Z 782.055,A -85,B 0,C 180,E1 17665.283,E2 17665.283} C_VEL
LIN {X 0,Y 505.982,Z 559.379,A -85,B 0,C 180,E1 17661.827,E2 17661.827} C_VEL
LIN {X 0,Y 508.306,Z 528.984,A -85,B 0,C 180,E1 17661.341,E2 17661.341} C_VEL
LIN {X 0,Y 501.285,Z 517.9,A -85,B 0,C 180,E1 17658.672,E2 17658.672} C_VEL
LIN {X 0,Y 495.515,Z 509.148,A -85,B 0,C 180,E1 17656.109,E2 17656.109} C_VEL
LIN {X 0,Y 492.189,Z 504.348,A -85,B 0,C 180,E1 17654.41,E2 17654.41} C_VEL
LIN {X 0,Y 489.239,Z 500.055,A -85,B 0,C 180,E1 17652.692,E2 17652.692} C_VEL
LIN {X 0,Y 486.131,Z 495.46,A -85,B 0,C 180,E1 17650.548,E2 17650.548} C_VEL
LIN {X 0,Y 483.249,Z 491.239,A -85,B 0,C 180,E1 17648.028,E2 17648.028} C_VEL
LIN {X 0,Y 482.639,Z 490.363,A -85,B 0,C 180,E1 17647.38,E2 17647.38} C_VEL
LIN {X 0,Y 479.962,Z 486.405,A -85,B 0,C 180,E1 17643.105,E2 17643.105} C_VEL
LIN {X 0,Y 479.707,Z 484.976,A -85,B 0,C 180,E1 17641.792,E2 17641.792} C_VEL
LIN {X 0,Y 479.766,Z 485.113,A -85,B 0,C 180,E1 17638.328,E2 17638.328} C_VEL
LIN {X 0,Y 481.555,Z 489.418,A -85,B 0,C 180,E1 17634.28,E2 17634.28} C_VEL
LIN {X 0,Y 483.209,Z 490.999,A -85,B 0,C 180,E1 17632.45,E2 17632.45} C_VEL
LIN {X 0,Y 486.044,Z 495.413,A -85,B 0,C 180,E1 17629.929,E2 17629.929} C_VEL
LIN {X 0,Y 487.317,Z 497.221,A -85,B 0,C 180,E1 17628.999,E2 17628.999} C_VEL
LIN {X 0,Y 490.478,Z 501.741,A -85,B 0,C 180,E1 17626.981,E2 17626.981} C_VEL
LIN {X 0,Y 494.469,Z 507.664,A -85,B 0,C 180,E1 17624.819,E2 17624.819} C_VEL
LIN {X 0,Y 500.602,Z 518.255,A -85,B 0,C 180,E1 17621.965,E2 17621.965} C_VEL
LIN {X 0,Y 506.234,Z 528.316,A -85,B 0,C 180,E1 17619.718,E2 17619.718} C_VEL
LIN {X 0,Y 508.404,Z 532.429,A -85,B 0,C 180,E1 17618.916,E2 17618.916} C_VEL
LIN {X 0,Y 491.696,Z 752.537,A -85,B 0,C 180,E1 17615.499,E2 17615.499} C_VEL
LIN {X 0,Y 486.434,Z 820.858,A -85,B 0,C 180,E1 17614.416,E2 17614.416} C_VEL
LIN {X 0,Y 482.625,Z 850.093,A -85,B 0,C 180,E1 17613.856,E2 17613.856} C_VEL
LIN {X 0,Y 478.282,Z 873.992,A -85,B 0,C 180,E1 17613.269,E2 17613.269} C_VEL
LIN {X 0,Y 473.764,Z 894.802,A -85,B 0,C 180,E1 17612.634,E2 17612.634} C_VEL
LIN {X 0,Y 468.787,Z 914.704,A -85,B 0,C 180,E1 17611.905,E2 17611.905} C_VEL
LIN {X 0,Y 462.962,Z 935.345,A -85,B 0,C 180,E1 17611.007,E2 17611.007} C_VEL
LIN {X 0,Y 455.064,Z 960.355,A -85,B 0,C 180,E1 17609.711,E2 17609.711} C_VEL
LIN {X 0,Y 446.456,Z 984.184,A -85,B 0,C 180,E1 17608.201,E2 17608.201} C_VEL
LIN {X 0,Y 439.088,Z 1003.019,A -85,B 0,C 180,E1 17606.808,E2 17606.808} C_VEL
LIN {X 0,Y 431.676,Z 1020.693,A -85,B 0,C 180,E1 17605.311,E2 17605.311} C_VEL
LIN {X 0,Y 423.191,Z 1039.812,A -85,B 0,C 180,E1 17603.447,E2 17603.447} C_VEL
LIN {X 0,Y 412.343,Z 1062.853,A -85,B 0,C 180,E1 17600.78,E2 17600.78} C_VEL
LIN {X 0,Y 404.225,Z 1079.27,A -85,B 0,C 180,E1 17598.545,E2 17598.545} C_VEL
LIN {X 0,Y 396.484,Z 1094.568,A -85,B 0,C 180,E1 17596.157,E2 17596.157} C_VEL
LIN {X 0,Y 388.999,Z 1109.202,A -85,B 0,C 180,E1 17593.539,E2 17593.539} C_VEL
LIN {X 0,Y 380.15,Z 1126.505,A -85,B 0,C 180,E1 17589.923,E2 17589.923} C_VEL
LIN {X 0,Y 373.456,Z 1139.694,A -85,B 0,C 180,E1 17586.658,E2 17586.658} C_VEL
LIN {X 0,Y 368.062,Z 1150.867,A -85,B 0,C 180,E1 17583.467,E2 17583.467} C_VEL
LIN {X 0,Y 363.547,Z 1160.764,A -85,B 0,C 180,E1 17580.219,E2 17580.219} C_VEL
LIN {X 0,Y 359.124,Z 1171.542,A -85,B 0,C 180,E1 17576.097,E2 17576.097} C_VEL
LIN {X 0,Y 355.825,Z 1180.696,A -85,B 0,C 180,E1 17571.772,E2 17571.772} C_VEL
LIN {X 0,Y 354.03,Z 1186.849,A -85,B 0,C 180,E1 17568.27,E2 17568.27} C_VEL
LIN {X 0,Y 352.938,Z 1191.678,A -85,B 0,C 180,E1 17564.939,E2 17564.939} C_VEL
LIN {X 0,Y 352.3,Z 1195.522,A -85,B 0,C 180,E1 17561.625,E2 17561.625} C_VEL
LIN {X 0,Y 352.041,Z 1198.402,A -85,B 0,C 180,E1 17558.329,E2 17558.329} C_VEL
LIN {X 0,Y 351.965,Z 1200.26,A -85,B 0,C 180,E1 17555.216,E2 17555.216} C_VEL
LIN {X 0,Y 351.96,Z 1201.27,A -85,B 0,C 180,E1 17552.116,E2 17552.116} C_VEL
LIN {X 0,Y 351.964,Z 1201.411,A -85,B 0,C 180,E1 17548.861,E2 17548.861} C_VEL
LIN {X 0,Y 351.956,Z 1200.611,A -85,B 0,C 180,E1 17545.601,E2 17545.601} C_VEL
LIN {X 0,Y 352.016,Z 1198.87,A -85,B 0,C 180,E1 17542.328,E2 17542.328} C_VEL
LIN {X 0,Y 352.229,Z 1196.179,A -85,B 0,C 180,E1 17539.036,E2 17539.036} C_VEL
LIN {X 0,Y 352.818,Z 1192.313,A -85,B 0,C 180,E1 17535.559,E2 17535.559} C_VEL
LIN {X 0,Y 353.821,Z 1187.628,A -85,B 0,C 180,E1 17532.23,E2 17532.23} C_VEL
LIN {X 0,Y 355.526,Z 1181.62,A -85,B 0,C 180,E1 17528.728,E2 17528.728} C_VEL
LIN {X 0,Y 358.006,Z 1174.38,A -85,B 0,C 180,E1 17525.191,E2 17525.191} C_VEL
LIN {X 0,Y 362.181,Z 1164.03,A -85,B 0,C 180,E1 17520.93,E2 17520.93} C_VEL
LIN {X 0,Y 367.578,Z 1151.9,A -85,B 0,C 180,E1 17516.856,E2 17516.856} C_VEL
LIN {X 0,Y 372.87,Z 1140.838,A -85,B 0,C 180,E1 17513.657,E2 17513.657} C_VEL
LIN {X 0,Y 379.111,Z 1128.41,A -85,B 0,C 180,E1 17510.535,E2 17510.535} C_VEL
LIN {X 0,Y 387.447,Z 1112.282,A -85,B 0,C 180,E1 17507.056,E2 17507.056} C_VEL
LIN {X 0,Y 396.046,Z 1095.362,A -85,B 0,C 180,E1 17503.986,E2 17503.986} C_VEL
LIN {X 0,Y 403.513,Z 1080.604,A -85,B 0,C 180,E1 17501.662,E2 17501.662} C_VEL
LIN {X 0,Y 411.068,Z 1065.335,A -85,B 0,C 180,E1 17499.552,E2 17499.552} C_VEL
LIN {X 0,Y 419.394,Z 1047.936,A -85,B 0,C 180,E1 17497.45,E2 17497.45} C_VEL
LIN {X 0,Y 429.949,Z 1024.603,A -85,B 0,C 180,E1 17495.057,E2 17495.057} C_VEL
LIN {X 0,Y 438.197,Z 1005.021,A -85,B 0,C 180,E1 17493.362,E2 17493.362} C_VEL
LIN {X 0,Y 445.296,Z 986.975,A -85,B 0,C 180,E1 17492.001,E2 17492.001} C_VEL
LIN {X 0,Y 452.445,Z 967.425,A -85,B 0,C 180,E1 17490.723,E2 17490.723} C_VEL
LIN {X 0,Y 459.955,Z 944.979,A -85,B 0,C 180,E1 17489.47,E2 17489.47} C_VEL
LIN {X 0,Y 467.677,Z 918.556,A -85,B 0,C 180,E1 17488.258,E2 17488.258} C_VEL
LIN {X 0,Y 473.183,Z 896.844,A -85,B 0,C 180,E1 17487.442,E2 17487.442} C_VEL
LIN {X 0,Y 477.832,Z 875.679,A -85,B 0,C 180,E1 17486.785,E2 17486.785} C_VEL
LIN {X 0,Y 481.821,Z 854.129,A -85,B 0,C 180,E1 17486.242,E2 17486.242} C_VEL
LIN {X 0,Y 485.769,Z 826.778,A -85,B 0,C 180,E1 17485.691,E2 17485.691} C_VEL
LIN {X 0,Y 489.383,Z 782.485,A -85,B 0,C 180,E1 17484.975,E2 17484.975} C_VEL
LIN {X 0,Y 505.976,Z 561.83,A -85,B 0,C 180,E1 17481.545,E2 17481.545} C_VEL
LIN {X 0,Y 508.249,Z 532.077,A -85,B 0,C 180,E1 17481.071,E2 17481.071} C_VEL
LIN {X 0,Y 501.182,Z 519.374,A -85,B 0,C 180,E1 17478.344,E2 17478.344} C_VEL
LIN {X 0,Y 495.135,Z 509.063,A -85,B 0,C 180,E1 17475.61,E2 17475.61} C_VEL
LIN {X 0,Y 492.442,Z 504.748,A -85,B 0,C 180,E1 17474.223,E2 17474.223} C_VEL
LIN {X 0,Y 489.061,Z 499.819,A -85,B 0,C 180,E1 17472.277,E2 17472.277} C_VEL
LIN {X 0,Y 486.17,Z 495.578,A -85,B 0,C 180,E1 17470.308,E2 17470.308} C_VEL
LIN {X 0,Y 483.274,Z 491.374,A -85,B 0,C 180,E1 17467.849,E2 17467.849} C_VEL
LIN {X 0,Y 482.708,Z 490.447,A -85,B 0,C 180,E1 17467.259,E2 17467.259} C_VEL
LIN {X 0,Y 480.059,Z 487.038,A -85,B 0,C 180,E1 17463.583,E2 17463.583} C_VEL
LIN {X 0,Y 479.513,Z 484.933,A -85,B 0,C 180,E1 17461.673,E2 17461.673} C_VEL
LIN {X 0,Y 479.6,Z 485.041,A -85,B 0,C 180,E1 17457.491,E2 17457.491} C_VEL
LIN {X 0,Y 481.131,Z 488.995,A -85,B 0,C 180,E1 17454.036,E2 17454.036} C_VEL
LIN {X 0,Y 483.02,Z 490.918,A -85,B 0,C 180,E1 17451.908,E2 17451.908} C_VEL
LIN {X 0,Y 485.814,Z 495.184,A -85,B 0,C 180,E1 17449.445,E2 17449.445} C_VEL
LIN {X 0,Y 487.005,Z 496.892,A -85,B 0,C 180,E1 17448.572,E2 17448.572} C_VEL
LIN {X 0,Y 490.545,Z 502.016,A -85,B 0,C 180,E1 17446.323,E2 17446.323} C_VEL
LIN {X 0,Y 494.149,Z 507.248,A -85,B 0,C 180,E1 17444.388,E2 17444.388} C_VEL
LIN {X 0,Y 499.431,Z 515.104,A -85,B 0,C 180,E1 17441.952,E2 17441.952} C_VEL
LIN {X 0,Y 505.704,Z 525.034,A -85,B 0,C 180,E1 17439.454,E2 17439.454} C_VEL
LIN {X 0,Y 508.197,Z 529.232,A -85,B 0,C 180,E1 17438.545,E2 17438.545} C_VEL
LIN {X 0,Y 491.743,Z 745.221,A -85,B 0,C 180,E1 17435.194,E2 17435.194} C_VEL
LIN {X 0,Y 486.885,Z 807.435,A -85,B 0,C 180,E1 17434.209,E2 17434.209} C_VEL
LIN {X 0,Y 482.987,Z 837.207,A -85,B 0,C 180,E1 17433.619,E2 17433.619} C_VEL
LIN {X 0,Y 478.929,Z 860.133,A -85,B 0,C 180,E1 17433.014,E2 17433.014} C_VEL
LIN {X 0,Y 474.45,Z 881.137,A -85,B 0,C 180,E1 17432.336,E2 17432.336} C_VEL
LIN {X 0,Y 469.2,Z 902.341,A -85,B 0,C 180,E1 17431.513,E2 17431.513} C_VEL
LIN {X 0,Y 462.006,Z 927.68,A -85,B 0,C 180,E1 17430.332,E2 17430.332} C_VEL
LIN {X 0,Y 454.27,Z 951.049,A -85,B 0,C 180,E1 17428.999,E2 17428.999} C_VEL
LIN {X 0,Y 447.429,Z 969.775,A -85,B 0,C 180,E1 17427.76,E2 17427.76} C_VEL
LIN {X 0,Y 440.003,Z 988.563,A -85,B 0,C 180,E1 17426.325,E2 17426.325} C_VEL
LIN {X 0,Y 432.31,Z 1006.711,A -85,B 0,C 180,E1 17424.729,E2 17424.729} C_VEL
LIN {X 0,Y 422.697,Z 1027.954,A -85,B 0,C 180,E1 17422.559,E2 17422.559} C_VEL
LIN {X 0,Y 413.2,Z 1047.349,A -85,B 0,C 180,E1 17420.2,E2 17420.2} C_VEL
LIN {X 0,Y 405.496,Z 1062.521,A -85,B 0,C 180,E1 17418.068,E2 17418.068} C_VEL
LIN {X 0,Y 397.91,Z 1077.038,A -85,B 0,C 180,E1 17415.737,E2 17415.737} C_VEL
LIN {X 0,Y 389.602,Z 1092.658,A -85,B 0,C 180,E1 17412.85,E2 17412.85} C_VEL
LIN {X 0,Y 380.767,Z 1108.983,A -85,B 0,C 180,E1 17409.26,E2 17409.26} C_VEL
LIN {X 0,Y 374.414,Z 1120.926,A -85,B 0,C 180,E1 17406.169,E2 17406.169} C_VEL
LIN {X 0,Y 368.919,Z 1131.521,A -85,B 0,C 180,E1 17403.008,E2 17403.008} C_VEL
LIN {X 0,Y 363.521,Z 1142.652,A -85,B 0,C 180,E1 17399.133,E2 17399.133} C_VEL
LIN {X 0,Y 358.998,Z 1152.665,A -85,B 0,C 180,E1 17394.87,E2 17394.87} C_VEL
LIN {X 0,Y 356.238,Z 1159.692,A -85,B 0,C 180,E1 17391.273,E2 17391.273} C_VEL
LIN {X 0,Y 354.404,Z 1165.18,A -85,B 0,C 180,E1 17387.909,E2 17387.909} C_VEL
LIN {X 0,Y 353.169,Z 1169.818,A -85,B 0,C 180,E1 17384.426,E2 17384.426} C_VEL
LIN {X 0,Y 352.429,Z 1173.583,A -85,B 0,C 180,E1 17380.792,E2 17380.792} C_VEL
LIN {X 0,Y 352.075,Z 1176.593,A -85,B 0,C 180,E1 17376.686,E2 17376.686} C_VEL
LIN {X 0,Y 351.969,Z 1178.11,A -85,B 0,C 180,E1 17372.605,E2 17372.605} C_VEL
LIN {X 0,Y 351.961,Z 1178.34,A -85,B 0,C 180,E1 17369.023,E2 17369.023} C_VEL
LIN {X 0,Y 351.993,Z 1177.594,A -85,B 0,C 180,E1 17365.601,E2 17365.601} C_VEL
LIN {X 0,Y 352.115,Z 1175.998,A -85,B 0,C 180,E1 17362.329,E2 17362.329} C_VEL
LIN {X 0,Y 352.46,Z 1173.366,A -85,B 0,C 180,E1 17358.878,E2 17358.878} C_VEL
LIN {X 0,Y 353.194,Z 1169.734,A -85,B 0,C 180,E1 17355.407,E2 17355.407} C_VEL
LIN {X 0,Y 354.434,Z 1165.096,A -85,B 0,C 180,E1 17351.937,E2 17351.937} C_VEL
LIN {X 0,Y 356.376,Z 1159.351,A -85,B 0,C 180,E1 17348.436,E2 17348.436} C_VEL
LIN {X 0,Y 359.541,Z 1151.488,A -85,B 0,C 180,E1 17344.466,E2 17344.466} C_VEL
LIN {X 0,Y 362.814,Z 1144.143,A -85,B 0,C 180,E1 17341.355,E2 17341.355} C_VEL
LIN {X 0,Y 363.232,Z 1141.49,A -85,B 0,C 180,E1 17340.205,E2 17340.205} C_VEL
LIN {X 0,Y 361.329,Z 1134.302,A -85,B 0,C 180,E1 17337.057,E2 17337.057} C_VEL
LIN {X 0,Y 362.102,Z 1131.565,A -85,B 0,C 180,E1 17336.1,E2 17336.1} C_VEL
LIN {X 0,Y 367.861,Z 1120.936,A -85,B 0,C 180,E1 17332.886,E2 17332.886} C_VEL
LIN {X 0,Y 374.542,Z 1108.963,A -85,B 0,C 180,E1 17329.757,E2 17329.757} C_VEL
LIN {X 0,Y 384.194,Z 1091.814,A -85,B 0,C 180,E1 17325.984,E2 17325.984} C_VEL
LIN {X 0,Y 392.194,Z 1077.349,A -85,B 0,C 180,E1 17323.3,E2 17323.3} C_VEL
LIN {X 0,Y 399.963,Z 1062.992,A -85,B 0,C 180,E1 17320.978,E2 17320.978} C_VEL
LIN {X 0,Y 408.182,Z 1047.335,A -85,B 0,C 180,E1 17318.771,E2 17318.771} C_VEL
LIN {X 0,Y 418.294,Z 1027.286,A -85,B 0,C 180,E1 17316.338,E2 17316.338} C_VEL
LIN {X 0,Y 427.573,Z 1007.307,A -85,B 0,C 180,E1 17314.304,E2 17314.304} C_VEL
LIN {X 0,Y 435.489,Z 989.145,A -85,B 0,C 180,E1 17312.705,E2 17312.705} C_VEL
LIN {X 0,Y 442.927,Z 970.823,A -85,B 0,C 180,E1 17311.304,E2 17311.304} C_VEL
LIN {X 0,Y 449.972,Z 952.052,A -85,B 0,C 180,E1 17310.062,E2 17310.062} C_VEL
LIN {X 0,Y 457.504,Z 929.883,A -85,B 0,C 180,E1 17308.793,E2 17308.793} C_VEL
LIN {X 0,Y 465.239,Z 903.673,A -85,B 0,C 180,E1 17307.562,E2 17307.562} C_VEL
LIN {X 0,Y 470.72,Z 882.106,A -85,B 0,C 180,E1 17306.724,E2 17306.724} C_VEL
LIN {X 0,Y 475.289,Z 861.233,A -85,B 0,C 180,E1 17306.051,E2 17306.051} C_VEL
LIN {X 0,Y 479.23,Z 839.634,A -85,B 0,C 180,E1 17305.478,E2 17305.478} C_VEL
LIN {X 0,Y 483.149,Z 812.183,A -85,B 0,C 180,E1 17304.914,E2 17304.914} C_VEL
LIN {X 0,Y 486.939,Z 766.919,A -85,B 0,C 180,E1 17304.189,E2 17304.189} C_VEL
LIN {X 0,Y 504.275,Z 544.341,A -85,B 0,C 180,E1 17300.742,E2 17300.742} C_VEL
LIN {X 0,Y 505.049,Z 534.221,A -85,B 0,C 180,E1 17300.574,E2 17300.574} C_VEL
LIN {X 0,Y 498.313,Z 523.442,A -85,B 0,C 180,E1 17297.879,E2 17297.879} C_VEL
LIN {X 0,Y 493.26,Z 515.713,A -85,B 0,C 180,E1 17295.52,E2 17295.52} C_VEL
LIN {X 0,Y 490.579,Z 511.758,A -85,B 0,C 180,E1 17294.097,E2 17294.097} C_VEL
LIN {X 0,Y 487.889,Z 507.748,A -85,B 0,C 180,E1 17292.487,E2 17292.487} C_VEL
LIN {X 0,Y 484.843,Z 503.188,A -85,B 0,C 180,E1 17290.336,E2 17290.336} C_VEL
LIN {X 0,Y 482.046,Z 498.928,A -85,B 0,C 180,E1 17287.809,E2 17287.809} C_VEL
LIN {X 0,Y 481.119,Z 497.919,A -85,B 0,C 180,E1 17286.803,E2 17286.803} C_VEL
LIN {X 0,Y 478.891,Z 493.981,A -85,B 0,C 180,E1 17282.753,E2 17282.753} C_VEL
LIN {X 0,Y 478.733,Z 492.917,A -85,B 0,C 180,E1 17281.795,E2 17281.795} C_VEL
LIN {X 0,Y 478.779,Z 493.154,A -85,B 0,C 180,E1 17278.325,E2 17278.325} C_VEL
LIN {X 0,Y 480.58,Z 497.391,A -85,B 0,C 180,E1 17274.268,E2 17274.268} C_VEL
LIN {X 0,Y 482.109,Z 498.933,A -85,B 0,C 180,E1 17272.552,E2 17272.552} C_VEL
LIN {X 0,Y 484.914,Z 503.295,A -85,B 0,C 180,E1 17270.026,E2 17270.026} C_VEL
LIN {X 0,Y 486.489,Z 505.716,A -85,B 0,C 180,E1 17268.86,E2 17268.86} C_VEL
LIN {X 0,Y 489.102,Z 509.447,A -85,B 0,C 180,E1 17267.185,E2 17267.185} C_VEL
LIN {X 0,Y 492.807,Z 515.033,A -85,B 0,C 180,E1 17265.128,E2 17265.128} C_VEL
LIN {X 0,Y 498.745,Z 525.51,A -85,B 0,C 180,E1 17262.288,E2 17262.288} C_VEL
LIN {X 0,Y 504.194,Z 535.467,A -85,B 0,C 180,E1 17260.056,E2 17260.056} C_VEL
LIN {X 0,Y 505.137,Z 537.461,A -85,B 0,C 180,E1 17259.687,E2 17259.687} C_VEL
LIN {X 0,Y 488.016,Z 757.528,A -85,B 0,C 180,E1 17256.277,E2 17256.277} C_VEL
LIN {X 0,Y 482.977,Z 820.978,A -85,B 0,C 180,E1 17255.271,E2 17255.271} C_VEL
LIN {X 0,Y 478.923,Z 851.017,A -85,B 0,C 180,E1 17254.695,E2 17254.695} C_VEL
LIN {X 0,Y 474.613,Z 874.178,A -85,B 0,C 180,E1 17254.127,E2 17254.127} C_VEL
LIN {X 0,Y 469.878,Z 895.456,A -85,B 0,C 180,E1 17253.481,E2 17253.481} C_VEL
LIN {X 0,Y 464.467,Z 916.481,A -85,B 0,C 180,E1 17252.707,E2 17252.707} C_VEL
LIN {X 0,Y 457.032,Z 941.89,A -85,B 0,C 180,E1 17251.577,E2 17251.577} C_VEL
LIN {X 0,Y 448.755,Z 966.173,A -85,B 0,C 180,E1 17250.247,E2 17250.247} C_VEL
LIN {X 0,Y 441.529,Z 985.555,A -85,B 0,C 180,E1 17248.995,E2 17248.995} C_VEL
LIN {X 0,Y 434.303,Z 1003.493,A -85,B 0,C 180,E1 17247.662,E2 17247.662} C_VEL
LIN {X 0,Y 426.409,Z 1021.773,A -85,B 0,C 180,E1 17246.106,E2 17246.106} C_VEL
LIN {X 0,Y 416.326,Z 1043.831,A -85,B 0,C 180,E1 17243.915,E2 17243.915} C_VEL
LIN {X 0,Y 406.291,Z 1064.151,A -85,B 0,C 180,E1 17241.491,E2 17241.491} C_VEL
LIN {X 0,Y 398.213,Z 1079.935,A -85,B 0,C 180,E1 17239.313,E2 17239.313} C_VEL
LIN {X 0,Y 390.235,Z 1095.152,A -85,B 0,C 180,E1 17236.905,E2 17236.905} C_VEL
LIN {X 0,Y 381.308,Z 1112.061,A -85,B 0,C 180,E1 17233.809,E2 17233.809} C_VEL
LIN {X 0,Y 372.634,Z 1128.172,A -85,B 0,C 180,E1 17230.29,E2 17230.29} C_VEL
LIN {X 0,Y 366.097,Z 1140.589,A -85,B 0,C 180,E1 17227.127,E2 17227.127} C_VEL
LIN {X 0,Y 360.532,Z 1151.644,A -85,B 0,C 180,E1 17223.878,E2 17223.878} C_VEL
LIN {X 0,Y 354.852,Z 1163.773,A -85,B 0,C 180,E1 17219.73,E2 17219.73} C_VEL
LIN {X 0,Y 350.547,Z 1173.846,A -85,B 0,C 180,E1 17215.512,E2 17215.512} C_VEL
LIN {X 0,Y 347.898,Z 1181.048,A -85,B 0,C 180,E1 17211.939,E2 17211.939} C_VEL
LIN {X 0,Y 346.051,Z 1187.104,A -85,B 0,C 180,E1 17208.357,E2 17208.357} C_VEL
LIN {X 0,Y 344.893,Z 1192.051,A -85,B 0,C 180,E1 17204.78,E2 17204.78} C_VEL
LIN {X 0,Y 344.237,Z 1196.084,A -85,B 0,C 180,E1 17201.052,E2 17201.052} C_VEL
LIN {X 0,Y 343.987,Z 1199.315,A -85,B 0,C 180,E1 17196.844,E2 17196.844} C_VEL
LIN {X 0,Y 343.965,Z 1200.935,A -85,B 0,C 180,E1 17192.666,E2 17192.666} C_VEL
LIN {X 0,Y 343.965,Z 1201.172,A -85,B 0,C 180,E1 17189.001,E2 17189.001} C_VEL
LIN {X 0,Y 343.959,Z 1200.408,A -85,B 0,C 180,E1 17185.641,E2 17185.641} C_VEL
LIN {X 0,Y 344.022,Z 1198.604,A -85,B 0,C 180,E1 17182.149,E2 17182.149} C_VEL
LIN {X 0,Y 344.253,Z 1195.911,A -85,B 0,C 180,E1 17178.779,E2 17178.779} C_VEL
LIN {X 0,Y 344.893,Z 1192.044,A -85,B 0,C 180,E1 17175.22,E2 17175.22} C_VEL
LIN {X 0,Y 346.05,Z 1187.094,A -85,B 0,C 180,E1 17171.643,E2 17171.643} C_VEL
LIN {X 0,Y 347.804,Z 1181.317,A -85,B 0,C 180,E1 17168.215,E2 17168.215} C_VEL
LIN {X 0,Y 350.401,Z 1174.191,A -85,B 0,C 180,E1 17164.658,E2 17164.658} C_VEL
LIN {X 0,Y 354.651,Z 1164.177,A -85,B 0,C 180,E1 17160.438,E2 17160.438} C_VEL
LIN {X 0,Y 360.281,Z 1152.148,A -85,B 0,C 180,E1 17156.286,E2 17156.286} C_VEL
LIN {X 0,Y 365.79,Z 1141.145,A -85,B 0,C 180,E1 17153.033,E2 17153.033} C_VEL
LIN {X 0,Y 371.947,Z 1129.382,A -85,B 0,C 180,E1 17150.01,E2 17150.01} C_VEL
LIN {X 0,Y 379.482,Z 1115.326,A -85,B 0,C 180,E1 17146.875,E2 17146.875} C_VEL
LIN {X 0,Y 389.342,Z 1096.8,A -85,B 0,C 180,E1 17143.384,E2 17143.384} C_VEL
LIN {X 0,Y 397.481,Z 1081.265,A -85,B 0,C 180,E1 17140.896,E2 17140.896} C_VEL
LIN {X 0,Y 405.258,Z 1066.084,A -85,B 0,C 180,E1 17138.773,E2 17138.773} C_VEL
LIN {X 0,Y 413.259,Z 1049.906,A -85,B 0,C 180,E1 17136.79,E2 17136.79} C_VEL
LIN {X 0,Y 422.003,Z 1031.437,A -85,B 0,C 180,E1 17134.822,E2 17134.822} C_VEL
LIN {X 0,Y 432.449,Z 1007.774,A -85,B 0,C 180,E1 17132.691,E2 17132.691} C_VEL
LIN {X 0,Y 440.548,Z 987.821,A -85,B 0,C 180,E1 17131.171,E2 17131.171} C_VEL
LIN {X 0,Y 447.977,Z 968.057,A -85,B 0,C 180,E1 17129.876,E2 17129.876} C_VEL
LIN {X 0,Y 454.969,Z 947.74,A -85,B 0,C 180,E1 17128.735,E2 17128.735} C_VEL
LIN {X 0,Y 462.777,Z 922.425,A -85,B 0,C 180,E1 17127.541,E2 17127.541} C_VEL
LIN {X 0,Y 469.343,Z 897.237,A -85,B 0,C 180,E1 17126.587,E2 17126.587} C_VEL
LIN {X 0,Y 474.133,Z 875.948,A -85,B 0,C 180,E1 17125.929,E2 17125.929} C_VEL
LIN {X 0,Y 478.169,Z 854.673,A -85,B 0,C 180,E1 17125.395,E2 17125.395} C_VEL
LIN {X 0,Y 481.91,Z 829.646,A -85,B 0,C 180,E1 17124.888,E2 17124.888} C_VEL
LIN {X 0,Y 485.232,Z 792.918,A -85,B 0,C 180,E1 17124.28,E2 17124.28} C_VEL
LIN {X 0,Y 502.369,Z 570.361,A -85,B 0,C 180,E1 17120.826,E2 17120.826} C_VEL
LIN {X 0,Y 504.988,Z 537.131,A -85,B 0,C 180,E1 17120.304,E2 17120.304} C_VEL
LIN {X 0,Y 499.047,Z 526.185,A -85,B 0,C 180,E1 17117.912,E2 17117.912} C_VEL
LIN {X 0,Y 493.178,Z 515.915,A -85,B 0,C 180,E1 17115.162,E2 17115.162} C_VEL
LIN {X 0,Y 490.817,Z 512.159,A -85,B 0,C 180,E1 17113.91,E2 17113.91} C_VEL
LIN {X 0,Y 487.663,Z 507.454,A -85,B 0,C 180,E1 17112.043,E2 17112.043} C_VEL
LIN {X 0,Y 484.873,Z 503.301,A -85,B 0,C 180,E1 17110.095,E2 17110.095} C_VEL
LIN {X 0,Y 482.008,Z 498.937,A -85,B 0,C 180,E1 17107.569,E2 17107.569} C_VEL
LIN {X 0,Y 480.644,Z 497.481,A -85,B 0,C 180,E1 17106.09,E2 17106.09} C_VEL
LIN {X 0,Y 478.784,Z 494.025,A -85,B 0,C 180,E1 17102.753,E2 17102.753} C_VEL
LIN {X 0,Y 478.538,Z 492.874,A -85,B 0,C 180,E1 17101.676,E2 17101.676} C_VEL
LIN {X 0,Y 478.611,Z 493.106,A -85,B 0,C 180,E1 17097.485,E2 17097.485} C_VEL
LIN {X 0,Y 480.333,Z 497.197,A -85,B 0,C 180,E1 17093.786,E2 17093.786} C_VEL
LIN {X 0,Y 481.868,Z 498.733,A -85,B 0,C 180,E1 17092.068,E2 17092.068} C_VEL
LIN {X 0,Y 484.684,Z 503.067,A -85,B 0,C 180,E1 17089.54,E2 17089.54} C_VEL
LIN {X 0,Y 486.093,Z 505.284,A -85,B 0,C 180,E1 17088.491,E2 17088.491} C_VEL
LIN {X 0,Y 489.165,Z 509.719,A -85,B 0,C 180,E1 17086.525,E2 17086.525} C_VEL
LIN {X 0,Y 492.709,Z 514.968,A -85,B 0,C 180,E1 17084.583,E2 17084.583} C_VEL
LIN {X 0,Y 497.813,Z 522.728,A -85,B 0,C 180,E1 17082.181,E2 17082.181} C_VEL
LIN {X 0,Y 504.038,Z 532.763,A -85,B 0,C 180,E1 17079.656,E2 17079.656} C_VEL
LIN {X 0,Y 504.929,Z 534.425,A -85,B 0,C 180,E1 17079.315,E2 17079.315} C_VEL
LIN {X 0,Y 487.951,Z 751.927,A -85,B 0,C 180,E1 17075.947,E2 17075.947} C_VEL
LIN {X 0,Y 483.379,Z 808.522,A -85,B 0,C 180,E1 17075.05,E2 17075.05} C_VEL
LIN {X 0,Y 479.346,Z 838.263,A -85,B 0,C 180,E1 17074.458,E2 17074.458} C_VEL
LIN {X 0,Y 475.296,Z 860.624,A -85,B 0,C 180,E1 17073.87,E2 17073.87} C_VEL
LIN {X 0,Y 470.77,Z 881.411,A -85,B 0,C 180,E1 17073.203,E2 17073.203} C_VEL
LIN {X 0,Y 465.44,Z 902.487,A -85,B 0,C 180,E1 17072.391,E2 17072.391} C_VEL
LIN {X 0,Y 458.387,Z 926.884,A -85,B 0,C 180,E1 17071.266,E2 17071.266} C_VEL
LIN {X 0,Y 450.148,Z 951.297,A -85,B 0,C 180,E1 17069.887,E2 17069.887} C_VEL
LIN {X 0,Y 443.133,Z 970.048,A -85,B 0,C 180,E1 17068.652,E2 17068.652} C_VEL
LIN {X 0,Y 435.599,Z 988.66,A -85,B 0,C 180,E1 17067.234,E2 17067.234} C_VEL
LIN {X 0,Y 427.629,Z 1006.985,A -85,B 0,C 180,E1 17065.625,E2 17065.625} C_VEL
LIN {X 0,Y 417.934,Z 1027.859,A -85,B 0,C 180,E1 17063.498,E2 17063.498} C_VEL
LIN {X 0,Y 407.963,Z 1047.624,A -85,B 0,C 180,E1 17061.091,E2 17061.091} C_VEL
LIN {X 0,Y 400.153,Z 1062.529,A -85,B 0,C 180,E1 17058.991,E2 17058.991} C_VEL
LIN {X 0,Y 392.612,Z 1076.482,A -85,B 0,C 180,E1 17056.748,E2 17056.748} C_VEL
LIN {X 0,Y 384.944,Z 1090.353,A -85,B 0,C 180,E1 17054.2,E2 17054.2} C_VEL
LIN {X 0,Y 376.17,Z 1106.144,A -85,B 0,C 180,E1 17050.834,E2 17050.834} C_VEL
LIN {X 0,Y 368.314,Z 1120.081,A -85,B 0,C 180,E1 17047.256,E2 17047.256} C_VEL
LIN {X 0,Y 362.496,Z 1130.79,A -85,B 0,C 180,E1 17044.051,E2 17044.051} C_VEL
LIN {X 0,Y 357.553,Z 1140.242,A -85,B 0,C 180,E1 17040.78,E2 17040.78} C_VEL
LIN {X 0,Y 352.809,Z 1150.099,A -85,B 0,C 180,E1 17036.78,E2 17036.78} C_VEL
LIN {X 0,Y 348.883,Z 1159.168,A -85,B 0,C 180,E1 17032.224,E2 17032.224} C_VEL
LIN {X 0,Y 346.693,Z 1165.203,A -85,B 0,C 180,E1 17028.496,E2 17028.496} C_VEL
LIN {X 0,Y 345.324,Z 1169.887,A -85,B 0,C 180,E1 17024.933,E2 17024.933} C_VEL
LIN {X 0,Y 344.522,Z 1173.541,A -85,B 0,C 180,E1 17021.382,E2 17021.382} C_VEL
LIN {X 0,Y 344.139,Z 1176.199,A -85,B 0,C 180,E1 17017.848,E2 17017.848} C_VEL
LIN {X 0,Y 343.998,Z 1177.884,A -85,B 0,C 180,E1 17014.334,E2 17014.334} C_VEL
LIN {X 0,Y 343.959,Z 1178.656,A -85,B 0,C 180,E1 17010.5,E2 17010.5} C_VEL
LIN {X 0,Y 343.989,Z 1178.186,A -85,B 0,C 180,E1 17006.334,E2 17006.334} C_VEL
LIN {X 0,Y 344.124,Z 1176.373,A -85,B 0,C 180,E1 17002.319,E2 17002.319} C_VEL
LIN {X 0,Y 344.484,Z 1173.785,A -85,B 0,C 180,E1 16998.787,E2 16998.787} C_VEL
LIN {X 0,Y 345.254,Z 1170.201,A -85,B 0,C 180,E1 16995.235,E2 16995.235} C_VEL
LIN {X 0,Y 346.573,Z 1165.57,A -85,B 0,C 180,E1 16991.658,E2 16991.658} C_VEL
LIN {X 0,Y 348.596,Z 1159.915,A -85,B 0,C 180,E1 16988.107,E2 16988.107} C_VEL
LIN {X 0,Y 351.426,Z 1153.132,A -85,B 0,C 180,E1 16984.557,E2 16984.557} C_VEL
LIN {X 0,Y 356.169,Z 1143.171,A -85,B 0,C 180,E1 16980.206,E2 16980.206} C_VEL
LIN {X 0,Y 361.836,Z 1132.063,A -85,B 0,C 180,E1 16976.26,E2 16976.26} C_VEL
LIN {X 0,Y 362.102,Z 1131.565,A -85,B 0,C 180,E1 16976.1,E2 16976.1} C_VEL
LIN {X 0,Y 362.978,Z 1128.438,A -85,B 0,C 180,E1 16974.988,E2 16974.988} C_VEL
LIN {X 0,Y 362.42,Z 1120.272,A -85,B 0,C 180,E1 16971.886,E2 16971.886} C_VEL
LIN {X 0,Y 363.604,Z 1117.267,A -85,B 0,C 180,E1 16970.967,E2 16970.967} C_VEL
LIN {X 0,Y 372.063,Z 1102.666,A -85,B 0,C 180,E1 16967.374,E2 16967.374} C_VEL
LIN {X 0,Y 379.531,Z 1089.812,A -85,B 0,C 180,E1 16964.659,E2 16964.659} C_VEL
LIN {X 0,Y 387.336,Z 1076.204,A -85,B 0,C 180,E1 16962.158,E2 16962.158} C_VEL
LIN {X 0,Y 395.085,Z 1062.348,A -85,B 0,C 180,E1 16959.932,E2 16959.932} C_VEL
LIN {X 0,Y 403.559,Z 1046.684,A -85,B 0,C 180,E1 16957.734,E2 16957.734} C_VEL
LIN {X 0,Y 414.608,Z 1025.149,A -85,B 0,C 180,E1 16955.163,E2 16955.163} C_VEL
LIN {X 0,Y 423.458,Z 1006.581,A -85,B 0,C 180,E1 16953.295,E2 16953.295} C_VEL
LIN {X 0,Y 431.443,Z 988.681,A -85,B 0,C 180,E1 16951.733,E2 16951.733} C_VEL
LIN {X 0,Y 439.067,Z 970.282,A -85,B 0,C 180,E1 16950.337,E2 16950.337} C_VEL
LIN {X 0,Y 446.95,Z 949.633,A -85,B 0,C 180,E1 16948.992,E2 16948.992} C_VEL
LIN {X 0,Y 455.702,Z 923.698,A -85,B 0,C 180,E1 16947.574,E2 16947.574} C_VEL
LIN {X 0,Y 461.905,Z 902.653,A -85,B 0,C 180,E1 16946.621,E2 16946.621} C_VEL
LIN {X 0,Y 467.157,Z 882.36,A -85,B 0,C 180,E1 16945.843,E2 16945.843} C_VEL
LIN {X 0,Y 471.817,Z 861.485,A -85,B 0,C 180,E1 16945.175,E2 16945.175} C_VEL
LIN {X 0,Y 475.857,Z 839.754,A -85,B 0,C 180,E1 16944.603,E2 16944.603} C_VEL
LIN {X 0,Y 479.861,Z 812.103,A -85,B 0,C 180,E1 16944.042,E2 16944.042} C_VEL
LIN {X 0,Y 483.771,Z 766.394,A -85,B 0,C 180,E1 16943.312,E2 16943.312} C_VEL
LIN {X 0,Y 501.532,Z 544.093,A -85,B 0,C 180,E1 16939.878,E2 16939.878} C_VEL
LIN {X 0,Y 501.875,Z 539.527,A -85,B 0,C 180,E1 16939.797,E2 16939.797} C_VEL
LIN {X 0,Y 495.811,Z 529.53,A -85,B 0,C 180,E1 16937.245,E2 16937.245} C_VEL
LIN {X 0,Y 490.125,Z 520.672,A -85,B 0,C 180,E1 16934.412,E2 16934.412} C_VEL
LIN {X 0,Y 486.364,Z 515.213,A -85,B 0,C 180,E1 16932.165,E2 16932.165} C_VEL
LIN {X 0,Y 483.716,Z 511.07,A -85,B 0,C 180,E1 16930.24,E2 16930.24} C_VEL
LIN {X 0,Y 480.899,Z 506.74,A -85,B 0,C 180,E1 16927.647,E2 16927.647} C_VEL
LIN {X 0,Y 477.881,Z 501.863,A -85,B 0,C 180,E1 16922.638,E2 16922.638} C_VEL
LIN {X 0,Y 477.732,Z 500.854,A -85,B 0,C 180,E1 16921.679,E2 16921.679} C_VEL
LIN {X 0,Y 477.78,Z 501.035,A -85,B 0,C 180,E1 16918.441,E2 16918.441} C_VEL
LIN {X 0,Y 479.515,Z 505.273,A -85,B 0,C 180,E1 16914.376,E2 16914.376} C_VEL
LIN {X 0,Y 480.96,Z 506.743,A -85,B 0,C 180,E1 16912.714,E2 16912.714} C_VEL
LIN {X 0,Y 483.784,Z 511.177,A -85,B 0,C 180,E1 16910.122,E2 16910.122} C_VEL
LIN {X 0,Y 487.732,Z 517.15,A -85,B 0,C 180,E1 16907.389,E2 16907.389} C_VEL
LIN {X 0,Y 491.317,Z 522.685,A -85,B 0,C 180,E1 16905.353,E2 16905.353} C_VEL
LIN {X 0,Y 497.281,Z 533.44,A -85,B 0,C 180,E1 16902.446,E2 16902.446} C_VEL
LIN {X 0,Y 501.977,Z 542.318,A -85,B 0,C 180,E1 16900.471,E2 16900.471} C_VEL
LIN {X 0,Y 484.407,Z 762.774,A -85,B 0,C 180,E1 16897.063,E2 16897.063} C_VEL
LIN {X 0,Y 479.608,Z 821.315,A -85,B 0,C 180,E1 16896.135,E2 16896.135} C_VEL
LIN {X 0,Y 475.387,Z 851.597,A -85,B 0,C 180,E1 16895.554,E2 16895.554} C_VEL
LIN {X 0,Y 471.11,Z 874.086,A -85,B 0,C 180,E1 16895.007,E2 16895.007} C_VEL
LIN {X 0,Y 466.449,Z 894.667,A -85,B 0,C 180,E1 16894.388,E2 16894.388} C_VEL
LIN {X 0,Y 460.923,Z 915.755,A -85,B 0,C 180,E1 16893.624,E2 16893.624} C_VEL
LIN {X 0,Y 453.832,Z 939.569,A -85,B 0,C 180,E1 16892.582,E2 16892.582} C_VEL
LIN {X 0,Y 444.976,Z 965.278,A -85,B 0,C 180,E1 16891.202,E2 16891.202} C_VEL
LIN {X 0,Y 437.346,Z 985.29,A -85,B 0,C 180,E1 16889.919,E2 16889.919} C_VEL
LIN {X 0,Y 429.93,Z 1003.225,A -85,B 0,C 180,E1 16888.595,E2 16888.595} C_VEL
LIN {X 0,Y 421.613,Z 1021.989,A -85,B 0,C 180,E1 16886.999,E2 16886.999} C_VEL
LIN {X 0,Y 411.173,Z 1044.127,A -85,B 0,C 180,E1 16884.791,E2 16884.791} C_VEL
LIN {X 0,Y 401.134,Z 1063.849,A -85,B 0,C 180,E1 16882.433,E2 16882.433} C_VEL
LIN {X 0,Y 392.778,Z 1079.662,A -85,B 0,C 180,E1 16880.244,E2 16880.244} C_VEL
LIN {X 0,Y 384.518,Z 1094.877,A -85,B 0,C 180,E1 16877.824,E2 16877.824} C_VEL
LIN {X 0,Y 374.99,Z 1112.28,A -85,B 0,C 180,E1 16874.607,E2 16874.607} C_VEL
LIN {X 0,Y 366.062,Z 1128.196,A -85,B 0,C 180,E1 16871.071,E2 16871.071} C_VEL
LIN {X 0,Y 359.395,Z 1140.314,A -85,B 0,C 180,E1 16867.94,E2 16867.94} C_VEL
LIN {X 0,Y 353.543,Z 1151.368,A -85,B 0,C 180,E1 16864.642,E2 16864.642} C_VEL
LIN {X 0,Y 347.572,Z 1163.498,A -85,B 0,C 180,E1 16860.417,E2 16860.417} C_VEL
LIN {X 0,Y 343.01,Z 1173.572,A -85,B 0,C 180,E1 16856.114,E2 16856.114} C_VEL
LIN {X 0,Y 340.196,Z 1180.776,A -85,B 0,C 180,E1 16852.462,E2 16852.462} C_VEL
LIN {X 0,Y 338.276,Z 1186.624,A -85,B 0,C 180,E1 16848.937,E2 16848.937} C_VEL
LIN {X 0,Y 337.02,Z 1191.569,A -85,B 0,C 180,E1 16845.31,E2 16845.31} C_VEL
LIN {X 0,Y 336.325,Z 1195.32,A -85,B 0,C 180,E1 16841.837,E2 16841.837} C_VEL
LIN {X 0,Y 336.052,Z 1197.99,A -85,B 0,C 180,E1 16838.555,E2 16838.555} C_VEL
LIN {X 0,Y 335.971,Z 1199.804,A -85,B 0,C 180,E1 16835.293,E2 16835.293} C_VEL
LIN {X 0,Y 335.968,Z 1200.768,A -85,B 0,C 180,E1 16832.047,E2 16832.047} C_VEL
LIN {X 0,Y 335.972,Z 1200.886,A -85,B 0,C 180,E1 16828.806,E2 16828.806} C_VEL
LIN {X 0,Y 335.963,Z 1200.084,A -85,B 0,C 180,E1 16825.391,E2 16825.391} C_VEL
LIN {X 0,Y 336.031,Z 1198.339,A -85,B 0,C 180,E1 16821.961,E2 16821.961} C_VEL
LIN {X 0,Y 336.28,Z 1195.644,A -85,B 0,C 180,E1 16818.509,E2 16818.509} C_VEL
LIN {X 0,Y 336.975,Z 1191.774,A -85,B 0,C 180,E1 16814.864,E2 16814.864} C_VEL
LIN {X 0,Y 338.218,Z 1186.822,A -85,B 0,C 180,E1 16811.202,E2 16811.202} C_VEL
LIN {X 0,Y 340.083,Z 1181.073,A -85,B 0,C 180,E1 16807.712,E2 16807.712} C_VEL
LIN {X 0,Y 342.855,Z 1173.915,A -85,B 0,C 180,E1 16804.059,E2 16804.059} C_VEL
LIN {X 0,Y 347.422,Z 1163.775,A -85,B 0,C 180,E1 16799.702,E2 16799.702} C_VEL
LIN {X 0,Y 353.278,Z 1151.869,A -85,B 0,C 180,E1 16795.525,E2 16795.525} C_VEL
LIN {X 0,Y 359.072,Z 1140.866,A -85,B 0,C 180,E1 16792.222,E2 16792.222} C_VEL
LIN {X 0,Y 365.492,Z 1129.147,A -85,B 0,C 180,E1 16789.17,E2 16789.17} C_VEL
LIN {X 0,Y 373.178,Z 1115.366,A -85,B 0,C 180,E1 16786.057,E2 16786.057} C_VEL
LIN {X 0,Y 383.603,Z 1096.492,A -85,B 0,C 180,E1 16782.462,E2 16782.462} C_VEL
LIN {X 0,Y 392.265,Z 1080.516,A -85,B 0,C 180,E1 16779.895,E2 16779.895} C_VEL
LIN {X 0,Y 400.586,Z 1064.778,A -85,B 0,C 180,E1 16777.7,E2 16777.7} C_VEL
LIN {X 0,Y 409.443,Z 1047.381,A -85,B 0,C 180,E1 16775.592,E2 16775.592} C_VEL
LIN {X 0,Y 420.609,Z 1024.049,A -85,B 0,C 180,E1 16773.201,E2 16773.201} C_VEL
LIN {X 0,Y 429.285,Z 1004.531,A -85,B 0,C 180,E1 16771.52,E2 16771.52} C_VEL
LIN {X 0,Y 436.533,Z 987.073,A -85,B 0,C 180,E1 16770.213,E2 16770.213} C_VEL
LIN {X 0,Y 443.879,Z 967.957,A -85,B 0,C 180,E1 16768.968,E2 16768.968} C_VEL
LIN {X 0,Y 450.808,Z 948.304,A -85,B 0,C 180,E1 16767.868,E2 16767.868} C_VEL
LIN {X 0,Y 458.436,Z 924.306,A -85,B 0,C 180,E1 16766.731,E2 16766.731} C_VEL
LIN {X 0,Y 465.575,Z 897.779,A -85,B 0,C 180,E1 16765.723,E2 16765.723} C_VEL
LIN {X 0,Y 470.543,Z 876.217,A -85,B 0,C 180,E1 16765.059,E2 16765.059} C_VEL
LIN {X 0,Y 474.654,Z 855.04,A -85,B 0,C 180,E1 16764.53,E2 16764.53} C_VEL
LIN {X 0,Y 478.277,Z 831.521,A -85,B 0,C 180,E1 16764.055,E2 16764.055} C_VEL
LIN {X 0,Y 481.749,Z 795.566,A -85,B 0,C 180,E1 16763.453,E2 16763.453} C_VEL
LIN {X 0,Y 499.317,Z 573.045,A -85,B 0,C 180,E1 16760.008,E2 16760.008} C_VEL
LIN {X 0,Y 501.803,Z 542.076,A -85,B 0,C 180,E1 16759.517,E2 16759.517} C_VEL
LIN {X 0,Y 496.076,Z 531.381,A -85,B 0,C 180,E1 16757.084,E2 16757.084} C_VEL
LIN {X 0,Y 490.36,Z 521.188,A -85,B 0,C 180,E1 16754.224,E2 16754.224} C_VEL
LIN {X 0,Y 486.361,Z 515.199,A -85,B 0,C 180,E1 16751.864,E2 16751.864} C_VEL
LIN {X 0,Y 483.584,Z 511.023,A -85,B 0,C 180,E1 16749.882,E2 16749.882} C_VEL
LIN {X 0,Y 480.803,Z 506.624,A -85,B 0,C 180,E1 16747.348,E2 16747.348} C_VEL
LIN {X 0,Y 477.873,Z 502.343,A -85,B 0,C 180,E1 16742.998,E2 16742.998} C_VEL
LIN {X 0,Y 477.532,Z 500.806,A -85,B 0,C 180,E1 16741.56,E2 16741.56} C_VEL
LIN {X 0,Y 477.605,Z 500.993,A -85,B 0,C 180,E1 16737.6,E2 16737.6} C_VEL
LIN {X 0,Y 479.268,Z 505.077,A -85,B 0,C 180,E1 16733.892,E2 16733.892} C_VEL
LIN {X 0,Y 480.77,Z 506.67,A -85,B 0,C 180,E1 16732.17,E2 16732.17} C_VEL
LIN {X 0,Y 483.713,Z 511.11,A -85,B 0,C 180,E1 16729.519,E2 16729.519} C_VEL
LIN {X 0,Y 487.791,Z 517.422,A -85,B 0,C 180,E1 16726.727,E2 16726.727} C_VEL
LIN {X 0,Y 491.275,Z 522.687,A -85,B 0,C 180,E1 16724.778,E2 16724.778} C_VEL
LIN {X 0,Y 496.214,Z 530.366,A -85,B 0,C 180,E1 16722.407,E2 16722.407} C_VEL
LIN {X 0,Y 501.757,Z 539.466,A -85,B 0,C 180,E1 16720.099,E2 16720.099} C_VEL
LIN {X 0,Y 484.778,Z 751.769,A -85,B 0,C 180,E1 16716.818,E2 16716.818} C_VEL
LIN {X 0,Y 480.066,Z 808.718,A -85,B 0,C 180,E1 16715.918,E2 16715.918} C_VEL
LIN {X 0,Y 475.945,Z 838.54,A -85,B 0,C 180,E1 16715.329,E2 16715.329} C_VEL
LIN {X 0,Y 471.815,Z 860.899,A -85,B 0,C 180,E1 16714.745,E2 16714.745} C_VEL
LIN {X 0,Y 467.2,Z 881.684,A -85,B 0,C 180,E1 16714.083,E2 16714.083} C_VEL
LIN {X 0,Y 461.758,Z 902.76,A -85,B 0,C 180,E1 16713.278,E2 16713.278} C_VEL
LIN {X 0,Y 454.213,Z 928.225,A -85,B 0,C 180,E1 16712.106,E2 16712.106} C_VEL
LIN {X 0,Y 446.159,Z 951.48,A -85,B 0,C 180,E1 16710.795,E2 16710.795} C_VEL
LIN {X 0,Y 438.948,Z 970.321,A -85,B 0,C 180,E1 16709.56,E2 16709.56} C_VEL
LIN {X 0,Y 431.332,Z 988.705,A -85,B 0,C 180,E1 16708.165,E2 16708.165} C_VEL
LIN {X 0,Y 423.445,Z 1006.407,A -85,B 0,C 180,E1 16706.62,E2 16706.62} C_VEL
LIN {X 0,Y 414.003,Z 1026.248,A -85,B 0,C 180,E1 16704.62,E2 16704.62} C_VEL
LIN {X 0,Y 403.329,Z 1046.976,A -85,B 0,C 180,E1 16702.127,E2 16702.127} C_VEL
LIN {X 0,Y 395.165,Z 1062.087,A -85,B 0,C 180,E1 16700.006,E2 16700.006} C_VEL
LIN {X 0,Y 387.435,Z 1075.926,A -85,B 0,C 180,E1 16697.788,E2 16697.788} C_VEL
LIN {X 0,Y 379.703,Z 1089.424,A -85,B 0,C 180,E1 16695.315,E2 16695.315} C_VEL
LIN {X 0,Y 371.836,Z 1102.998,A -85,B 0,C 180,E1 16692.449,E2 16692.449} C_VEL
LIN {X 0,Y 362.708,Z 1118.673,A -85,B 0,C 180,E1 16688.536,E2 16688.536} C_VEL
LIN {X 0,Y 356.166,Z 1130.061,A -85,B 0,C 180,E1 16685.134,E2 16685.134} C_VEL
LIN {X 0,Y 350.907,Z 1139.622,A -85,B 0,C 180,E1 16681.812,E2 16681.812} C_VEL
LIN {X 0,Y 346.364,Z 1148.396,A -85,B 0,C 180,E1 16678.257,E2 16678.257} C_VEL
LIN {X 0,Y 342.077,Z 1157.665,A -85,B 0,C 180,E1 16673.788,E2 16673.788} C_VEL
LIN {X 0,Y 339.092,Z 1164.982,A -85,B 0,C 180,E1 16669.284,E2 16669.284} C_VEL
LIN {X 0,Y 337.553,Z 1169.757,A -85,B 0,C 180,E1 16665.637,E2 16665.637} C_VEL
LIN {X 0,Y 336.63,Z 1173.501,A -85,B 0,C 180,E1 16662,E2 16662} C_VEL
LIN {X 0,Y 336.207,Z 1176.136,A -85,B 0,C 180,E1 16658.551,E2 16658.551} C_VEL
LIN {X 0,Y 336.025,Z 1177.821,A -85,B 0,C 180,E1 16655.293,E2 16655.293} C_VEL
LIN {X 0,Y 335.974,Z 1178.721,A -85,B 0,C 180,E1 16652.047,E2 16652.047} C_VEL
LIN {X 0,Y 335.974,Z 1178.82,A -85,B 0,C 180,E1 16648.636,E2 16648.636} C_VEL
LIN {X 0,Y 336.009,Z 1178.055,A -85,B 0,C 180,E1 16645.221,E2 16645.221} C_VEL
LIN {X 0,Y 336.167,Z 1176.418,A -85,B 0,C 180,E1 16641.792,E2 16641.792} C_VEL
LIN {X 0,Y 336.558,Z 1173.897,A -85,B 0,C 180,E1 16638.345,E2 16638.345} C_VEL
LIN {X 0,Y 337.417,Z 1170.268,A -85,B 0,C 180,E1 16634.709,E2 16634.709} C_VEL
LIN {X 0,Y 338.873,Z 1165.612,A -85,B 0,C 180,E1 16631.061,E2 16631.061} C_VEL
LIN {X 0,Y 341.067,Z 1159.891,A -85,B 0,C 180,E1 16627.416,E2 16627.416} C_VEL
LIN {X 0,Y 344.539,Z 1152.203,A -85,B 0,C 180,E1 16623.362,E2 16623.362} C_VEL
LIN {X 0,Y 349.853,Z 1141.651,A -85,B 0,C 180,E1 16618.85,E2 16618.85} C_VEL
LIN {X 0,Y 355.386,Z 1131.507,A -85,B 0,C 180,E1 16615.241,E2 16615.241} C_VEL
LIN {X 0,Y 361.246,Z 1121.182,A -85,B 0,C 180,E1 16612.078,E2 16612.078} C_VEL
LIN {X 0,Y 363.604,Z 1117.267,A -85,B 0,C 180,E1 16610.967,E2 16610.967} C_VEL
LIN {X 0,Y 364.959,Z 1113.705,A -85,B 0,C 180,E1 16609.902,E2 16609.902} C_VEL
LIN {X 0,Y 365.655,Z 1104.41,A -85,B 0,C 180,E1 16606.908,E2 16606.908} C_VEL
LIN {X 0,Y 367.14,Z 1100.966,A -85,B 0,C 180,E1 16606.045,E2 16606.045} C_VEL
LIN {X 0,Y 375.078,Z 1087.81,A -85,B 0,C 180,E1 16603.303,E2 16603.303} C_VEL
LIN {X 0,Y 385.19,Z 1070.792,A -85,B 0,C 180,E1 16600.257,E2 16600.257} C_VEL
LIN {X 0,Y 395.672,Z 1052.161,A -85,B 0,C 180,E1 16597.489,E2 16597.489} C_VEL
LIN {X 0,Y 404.346,Z 1036.067,A -85,B 0,C 180,E1 16595.435,E2 16595.435} C_VEL
LIN {X 0,Y 412.881,Z 1019.402,A -85,B 0,C 180,E1 16593.587,E2 16593.587} C_VEL
LIN {X 0,Y 421.811,Z 1000.899,A -85,B 0,C 180,E1 16591.812,E2 16591.812} C_VEL
LIN {X 0,Y 432.717,Z 976.174,A -85,B 0,C 180,E1 16589.814,E2 16589.814} C_VEL
LIN {X 0,Y 440.77,Z 955.975,A -85,B 0,C 180,E1 16588.45,E2 16588.45} C_VEL
LIN {X 0,Y 447.501,Z 937.386,A -85,B 0,C 180,E1 16587.36,E2 16587.36} C_VEL
LIN {X 0,Y 454.108,Z 917.218,A -85,B 0,C 180,E1 16586.346,E2 16586.346} C_VEL
LIN {X 0,Y 460.851,Z 893.967,A -85,B 0,C 180,E1 16585.361,E2 16585.361} C_VEL
LIN {X 0,Y 467.459,Z 866.489,A -85,B 0,C 180,E1 16584.424,E2 16584.424} C_VEL
LIN {X 0,Y 471.8,Z 844.418,A -85,B 0,C 180,E1 16583.825,E2 16583.825} C_VEL
LIN {X 0,Y 475.225,Z 822.824,A -85,B 0,C 180,E1 16583.357,E2 16583.357} C_VEL
LIN {X 0,Y 477.96,Z 799.313,A -85,B 0,C 180,E1 16582.947,E2 16582.947} C_VEL
LIN {X 0,Y 495.926,Z 579.411,A -85,B 0,C 180,E1 16579.552,E2 16579.552} C_VEL
LIN {X 0,Y 498.805,Z 544.744,A -85,B 0,C 180,E1 16579.011,E2 16579.011} C_VEL
LIN {X 0,Y 493.107,Z 535.467,A -85,B 0,C 180,E1 16576.492,E2 16576.492} C_VEL
LIN {X 0,Y 488.513,Z 528.098,A -85,B 0,C 180,E1 16574.097,E2 16574.097} C_VEL
LIN {X 0,Y 484.942,Z 522.788,A -85,B 0,C 180,E1 16571.899,E2 16571.899} C_VEL
LIN {X 0,Y 482.437,Z 518.795,A -85,B 0,C 180,E1 16570.026,E2 16570.026} C_VEL
LIN {X 0,Y 479.708,Z 514.43,A -85,B 0,C 180,E1 16567.425,E2 16567.425} C_VEL
LIN {X 0,Y 476.895,Z 509.897,A -85,B 0,C 180,E1 16562.644,E2 16562.644} C_VEL
LIN {X 0,Y 476.733,Z 508.791,A -85,B 0,C 180,E1 16561.562,E2 16561.562} C_VEL
LIN {X 0,Y 476.794,Z 509.07,A -85,B 0,C 180,E1 16558.438,E2 16558.438} C_VEL
LIN {X 0,Y 478.541,Z 513.246,A -85,B 0,C 180,E1 16554.364,E2 16554.364} C_VEL
LIN {X 0,Y 479.865,Z 514.672,A -85,B 0,C 180,E1 16552.818,E2 16552.818} C_VEL
LIN {X 0,Y 482.656,Z 519.058,A -85,B 0,C 180,E1 16550.219,E2 16550.219} C_VEL
LIN {X 0,Y 486.369,Z 524.851,A -85,B 0,C 180,E1 16547.594,E2 16547.594} C_VEL
LIN {X 0,Y 489.782,Z 530.252,A -85,B 0,C 180,E1 16545.608,E2 16545.608} C_VEL
LIN {X 0,Y 495.635,Z 541.027,A -85,B 0,C 180,E1 16542.688,E2 16542.688} C_VEL
LIN {X 0,Y 498.881,Z 547.535,A -85,B 0,C 180,E1 16541.259,E2 16541.259} C_VEL
LIN {X 0,Y 480.84,Z 768.658,A -85,B 0,C 180,E1 16537.851,E2 16537.851} C_VEL
LIN {X 0,Y 476.332,Z 821.823,A -85,B 0,C 180,E1 16537.008,E2 16537.008} C_VEL
LIN {X 0,Y 472.082,Z 851.507,A -85,B 0,C 180,E1 16536.44,E2 16536.44} C_VEL
LIN {X 0,Y 467.712,Z 874.027,A -85,B 0,C 180,E1 16535.898,E2 16535.898} C_VEL
LIN {X 0,Y 462.875,Z 894.94,A -85,B 0,C 180,E1 16535.274,E2 16535.274} C_VEL
LIN {X 0,Y 456.974,Z 916.916,A -85,B 0,C 180,E1 16534.48,E2 16534.48} C_VEL
LIN {X 0,Y 448.775,Z 943.403,A -85,B 0,C 180,E1 16533.305,E2 16533.305} C_VEL
LIN {X 0,Y 440.738,Z 965.922,A -85,B 0,C 180,E1 16532.082,E2 16532.082} C_VEL
LIN {X 0,Y 433.273,Z 985.038,A -85,B 0,C 180,E1 16530.86,E2 16530.86} C_VEL
LIN {X 0,Y 425.675,Z 1002.958,A -85,B 0,C 180,E1 16529.546,E2 16529.546} C_VEL
LIN {X 0,Y 417.059,Z 1021.91,A -85,B 0,C 180,E1 16527.938,E2 16527.938} C_VEL
LIN {X 0,Y 406.415,Z 1043.856,A -85,B 0,C 180,E1 16525.753,E2 16525.753} C_VEL
LIN {X 0,Y 396.074,Z 1063.577,A -85,B 0,C 180,E1 16523.395,E2 16523.395} C_VEL
LIN {X 0,Y 387.453,Z 1079.388,A -85,B 0,C 180,E1 16521.2,E2 16521.2} C_VEL
LIN {X 0,Y 378.91,Z 1094.603,A -85,B 0,C 180,E1 16518.768,E2 16518.768} C_VEL
LIN {X 0,Y 369.281,Z 1111.51,A -85,B 0,C 180,E1 16515.627,E2 16515.627} C_VEL
LIN {X 0,Y 359.905,Z 1127.62,A -85,B 0,C 180,E1 16512.03,E2 16512.03} C_VEL
LIN {X 0,Y 352.777,Z 1140.038,A -85,B 0,C 180,E1 16508.783,E2 16508.783} C_VEL
LIN {X 0,Y 346.625,Z 1151.092,A -85,B 0,C 180,E1 16505.436,E2 16505.436} C_VEL
LIN {X 0,Y 340.345,Z 1163.223,A -85,B 0,C 180,E1 16501.134,E2 16501.134} C_VEL
LIN {X 0,Y 335.51,Z 1173.299,A -85,B 0,C 180,E1 16496.743,E2 16496.743} C_VEL
LIN {X 0,Y 332.4,Z 1180.816,A -85,B 0,C 180,E1 16492.832,E2 16492.832} C_VEL
LIN {X 0,Y 330.379,Z 1186.624,A -85,B 0,C 180,E1 16489.218,E2 16489.218} C_VEL
LIN {X 0,Y 329.065,Z 1191.514,A -85,B 0,C 180,E1 16485.509,E2 16485.509} C_VEL
LIN {X 0,Y 328.314,Z 1195.385,A -85,B 0,C 180,E1 16481.773,E2 16481.773} C_VEL
LIN {X 0,Y 328.026,Z 1198.316,A -85,B 0,C 180,E1 16477.884,E2 16477.884} C_VEL
LIN {X 0,Y 327.964,Z 1200.247,A -85,B 0,C 180,E1 16473.671,E2 16473.671} C_VEL
LIN {X 0,Y 327.966,Z 1200.716,A -85,B 0,C 180,E1 16469.476,E2 16469.476} C_VEL
LIN {X 0,Y 327.965,Z 1199.921,A -85,B 0,C 180,E1 16465.526,E2 16465.526} C_VEL
LIN {X 0,Y 328.04,Z 1198.074,A -85,B 0,C 180,E1 16461.764,E2 16461.764} C_VEL
LIN {X 0,Y 328.314,Z 1195.377,A -85,B 0,C 180,E1 16458.226,E2 16458.226} C_VEL
LIN {X 0,Y 329.065,Z 1191.504,A -85,B 0,C 180,E1 16454.491,E2 16454.491} C_VEL
LIN {X 0,Y 330.397,Z 1186.55,A -85,B 0,C 180,E1 16450.74,E2 16450.74} C_VEL
LIN {X 0,Y 332.4,Z 1180.799,A -85,B 0,C 180,E1 16447.168,E2 16447.168} C_VEL
LIN {X 0,Y 335.508,Z 1173.276,A -85,B 0,C 180,E1 16443.256,E2 16443.256} C_VEL
LIN {X 0,Y 340.57,Z 1162.726,A -85,B 0,C 180,E1 16438.689,E2 16438.689} C_VEL
LIN {X 0,Y 346.624,Z 1151.063,A -85,B 0,C 180,E1 16434.564,E2 16434.564} C_VEL
LIN {X 0,Y 352.789,Z 1139.969,A -85,B 0,C 180,E1 16431.208,E2 16431.208} C_VEL
LIN {X 0,Y 359.901,Z 1127.572,A -85,B 0,C 180,E1 16427.969,E2 16427.969} C_VEL
LIN {X 0,Y 369.549,Z 1110.937,A -85,B 0,C 180,E1 16424.273,E2 16424.273} C_VEL
LIN {X 0,Y 378.899,Z 1094.523,A -85,B 0,C 180,E1 16421.23,E2 16421.23} C_VEL
LIN {X 0,Y 387.441,Z 1079.297,A -85,B 0,C 180,E1 16418.798,E2 16418.798} C_VEL
LIN {X 0,Y 396.307,Z 1063.02,A -85,B 0,C 180,E1 16416.544,E2 16416.544} C_VEL
LIN {X 0,Y 407.398,Z 1041.708,A -85,B 0,C 180,E1 16414.028,E2 16414.028} C_VEL
LIN {X 0,Y 417.354,Z 1021.073,A -85,B 0,C 180,E1 16411.997,E2 16411.997} C_VEL
LIN {X 0,Y 425.658,Z 1002.771,A -85,B 0,C 180,E1 16410.45,E2 16410.45} C_VEL
LIN {X 0,Y 433.197,Z 984.975,A -85,B 0,C 180,E1 16409.145,E2 16409.145} C_VEL
LIN {X 0,Y 441.066,Z 964.788,A -85,B 0,C 180,E1 16407.86,E2 16407.86} C_VEL
LIN {X 0,Y 450.175,Z 938.817,A -85,B 0,C 180,E1 16406.482,E2 16406.482} C_VEL
LIN {X 0,Y 457.083,Z 916.105,A -85,B 0,C 180,E1 16405.496,E2 16405.496} C_VEL
LIN {X 0,Y 462.854,Z 894.533,A -85,B 0,C 180,E1 16404.72,E2 16404.72} C_VEL
LIN {X 0,Y 467.691,Z 873.546,A -85,B 0,C 180,E1 16404.096,E2 16404.096} C_VEL
LIN {X 0,Y 472.244,Z 849.926,A -85,B 0,C 180,E1 16403.533,E2 16403.533} C_VEL
LIN {X 0,Y 476.344,Z 820.374,A -85,B 0,C 180,E1 16402.974,E2 16402.974} C_VEL
LIN {X 0,Y 481.854,Z 754.144,A -85,B 0,C 180,E1 16401.931,E2 16401.931} C_VEL
LIN {X 0,Y 498.741,Z 547.166,A -85,B 0,C 180,E1 16398.736,E2 16398.736} C_VEL
LIN {X 0,Y 493.545,Z 537.363,A -85,B 0,C 180,E1 16396.417,E2 16396.417} C_VEL
LIN {X 0,Y 488.432,Z 528.085,A -85,B 0,C 180,E1 16393.737,E2 16393.737} C_VEL
LIN {X 0,Y 484.843,Z 522.653,A -85,B 0,C 180,E1 16391.54,E2 16391.54} C_VEL
LIN {X 0,Y 482.302,Z 518.743,A -85,B 0,C 180,E1 16389.667,E2 16389.667} C_VEL
LIN {X 0,Y 479.328,Z 514.012,A -85,B 0,C 180,E1 16386.829,E2 16386.829} C_VEL
LIN {X 0,Y 476.928,Z 510.527,A -85,B 0,C 180,E1 16383.125,E2 16383.125} C_VEL
LIN {X 0,Y 476.528,Z 508.739,A -85,B 0,C 180,E1 16381.443,E2 16381.443} C_VEL
LIN {X 0,Y 476.601,Z 508.88,A -85,B 0,C 180,E1 16377.715,E2 16377.715} C_VEL
LIN {X 0,Y 478.293,Z 513.061,A -85,B 0,C 180,E1 16373.88,E2 16373.88} C_VEL
LIN {X 0,Y 479.624,Z 514.482,A -85,B 0,C 180,E1 16372.332,E2 16372.332} C_VEL
LIN {X 0,Y 483.095,Z 519.969,A -85,B 0,C 180,E1 16369.204,E2 16369.204} C_VEL
LIN {X 0,Y 486.516,Z 525.279,A -85,B 0,C 180,E1 16366.874,E2 16366.874} C_VEL
LIN {X 0,Y 489.847,Z 530.403,A -85,B 0,C 180,E1 16364.975,E2 16364.975} C_VEL
LIN {X 0,Y 494.956,Z 538.564,A -85,B 0,C 180,E1 16362.482,E2 16362.482} C_VEL
LIN {X 0,Y 498.657,Z 544.954,A -85,B 0,C 180,E1 16360.882,E2 16360.882} C_VEL
LIN {X 0,Y 480.421,Z 767.904,A -85,B 0,C 180,E1 16357.448,E2 16357.448} C_VEL
LIN {X 0,Y 476.459,Z 812.968,A -85,B 0,C 180,E1 16356.73,E2 16356.73} C_VEL
LIN {X 0,Y 472.403,Z 840.245,A -85,B 0,C 180,E1 16356.178,E2 16356.178} C_VEL
LIN {X 0,Y 468.309,Z 861.822,A -85,B 0,C 180,E1 16355.615,E2 16355.615} C_VEL
LIN {X 0,Y 463.543,Z 882.768,A -85,B 0,C 180,E1 16354.949,E2 16354.949} C_VEL
LIN {X 0,Y 457.837,Z 904.311,A -85,B 0,C 180,E1 16354.126,E2 16354.126} C_VEL
LIN {X 0,Y 449.748,Z 930.593,A -85,B 0,C 180,E1 16352.906,E2 16352.906} C_VEL
LIN {X 0,Y 441.914,Z 952.646,A -85,B 0,C 180,E1 16351.659,E2 16351.659} C_VEL
LIN {X 0,Y 434.547,Z 971.398,A -85,B 0,C 180,E1 16350.429,E2 16350.429} C_VEL
LIN {X 0,Y 426.76,Z 989.705,A -85,B 0,C 180,E1 16349.037,E2 16349.037} C_VEL
LIN {X 0,Y 418.285,Z 1008.193,A -85,B 0,C 180,E1 16347.416,E2 16347.416} C_VEL
LIN {X 0,Y 407.136,Z 1030.669,A -85,B 0,C 180,E1 16345.094,E2 16345.094} C_VEL
LIN {X 0,Y 397.797,Z 1048.173,A -85,B 0,C 180,E1 16342.942,E2 16342.942} C_VEL
LIN {X 0,Y 389.479,Z 1063.08,A -85,B 0,C 180,E1 16340.831,E2 16340.831} C_VEL
LIN {X 0,Y 381.411,Z 1077.033,A -85,B 0,C 180,E1 16338.568,E2 16338.568} C_VEL
LIN {X 0,Y 372.999,Z 1091.214,A -85,B 0,C 180,E1 16335.922,E2 16335.922} C_VEL
LIN {X 0,Y 363.323,Z 1107.32,A -85,B 0,C 180,E1 16332.395,E2 16332.395} C_VEL
LIN {X 0,Y 355.167,Z 1120.633,A -85,B 0,C 180,E1 16328.887,E2 16328.887} C_VEL
LIN {X 0,Y 348.778,Z 1131.342,A -85,B 0,C 180,E1 16325.588,E2 16325.588} C_VEL
LIN {X 0,Y 343.354,Z 1140.792,A -85,B 0,C 180,E1 16322.202,E2 16322.202} C_VEL
LIN {X 0,Y 338.077,Z 1150.641,A -85,B 0,C 180,E1 16318.05,E2 16318.05} C_VEL
LIN {X 0,Y 333.657,Z 1159.704,A -85,B 0,C 180,E1 16313.301,E2 16313.301} C_VEL
LIN {X 0,Y 331.246,Z 1165.499,A -85,B 0,C 180,E1 16309.576,E2 16309.576} C_VEL
LIN {X 0,Y 329.631,Z 1170.225,A -85,B 0,C 180,E1 16305.842,E2 16305.842} C_VEL
LIN {X 0,Y 328.696,Z 1173.768,A -85,B 0,C 180,E1 16302.294,E2 16302.294} C_VEL
LIN {X 0,Y 328.233,Z 1176.401,A -85,B 0,C 180,E1 16298.761,E2 16298.761} C_VEL
LIN {X 0,Y 328.036,Z 1178.084,A -85,B 0,C 180,E1 16295.422,E2 16295.422} C_VEL
LIN {X 0,Y 327.979,Z 1178.984,A -85,B 0,C 180,E1 16292.096,E2 16292.096} C_VEL
LIN {X 0,Y 327.978,Z 1179.105,A -85,B 0,C 180,E1 16288.777,E2 16288.777} C_VEL
LIN {X 0,Y 328.014,Z 1178.383,A -85,B 0,C 180,E1 16285.279,E2 16285.279} C_VEL
LIN {X 0,Y 328.196,Z 1176.682,A -85,B 0,C 180,E1 16281.591,E2 16281.591} C_VEL
LIN {X 0,Y 328.616,Z 1174.163,A -85,B 0,C 180,E1 16278.059,E2 16278.059} C_VEL
LIN {X 0,Y 329.544,Z 1170.536,A -85,B 0,C 180,E1 16274.334,E2 16274.334} C_VEL
LIN {X 0,Y 331.111,Z 1165.881,A -85,B 0,C 180,E1 16270.6,E2 16270.6} C_VEL
LIN {X 0,Y 333.453,Z 1160.161,A -85,B 0,C 180,E1 16266.871,E2 16266.871} C_VEL
LIN {X 0,Y 337.044,Z 1152.645,A -85,B 0,C 180,E1 16262.816,E2 16262.816} C_VEL
LIN {X 0,Y 342.835,Z 1141.774,A -85,B 0,C 180,E1 16258.072,E2 16258.072} C_VEL
LIN {X 0,Y 348.364,Z 1132.104,A -85,B 0,C 180,E1 16254.566,E2 16254.566} C_VEL
LIN {X 0,Y 354.677,Z 1121.481,A -85,B 0,C 180,E1 16251.257,E2 16251.257} C_VEL
LIN {X 0,Y 362.222,Z 1109.105,A -85,B 0,C 180,E1 16247.95,E2 16247.95} C_VEL
LIN {X 0,Y 367.14,Z 1100.966,A -85,B 0,C 180,E1 16246.045,E2 16246.045} C_VEL
LIN {X 0,Y 368.875,Z 1097.007,A -85,B 0,C 180,E1 16245.042,E2 16245.042} C_VEL
LIN {X 0,Y 370.886,Z 1086.767,A -85,B 0,C 180,E1 16242.174,E2 16242.174} C_VEL
LIN {X 0,Y 372.671,Z 1082.974,A -85,B 0,C 180,E1 16241.378,E2 16241.378} C_VEL
LIN {X 0,Y 383.045,Z 1065.624,A -85,B 0,C 180,E1 16238.456,E2 16238.456} C_VEL
LIN {X 0,Y 391.832,Z 1050.428,A -85,B 0,C 180,E1 16236.259,E2 16236.259} C_VEL
LIN {X 0,Y 400.518,Z 1034.688,A -85,B 0,C 180,E1 16234.279,E2 16234.279} C_VEL
LIN {X 0,Y 410.262,Z 1016.059,A -85,B 0,C 180,E1 16232.255,E2 16232.255} C_VEL
LIN {X 0,Y 421.437,Z 992.847,A -85,B 0,C 180,E1 16230.143,E2 16230.143} C_VEL
LIN {X 0,Y 430.053,Z 973.219,A -85,B 0,C 180,E1 16228.637,E2 16228.637} C_VEL
LIN {X 0,Y 437.576,Z 954.621,A -85,B 0,C 180,E1 16227.412,E2 16227.412} C_VEL
LIN {X 0,Y 444.891,Z 934.652,A -85,B 0,C 180,E1 16226.27,E2 16226.27} C_VEL
LIN {X 0,Y 453.11,Z 909.576,A -85,B 0,C 180,E1 16225.068,E2 16225.068} C_VEL
LIN {X 0,Y 460.005,Z 884.342,A -85,B 0,C 180,E1 16224.091,E2 16224.091} C_VEL
LIN {X 0,Y 464.943,Z 863.245,A -85,B 0,C 180,E1 16223.421,E2 16223.421} C_VEL
LIN {X 0,Y 469.081,Z 842.069,A -85,B 0,C 180,E1 16222.866,E2 16222.866} C_VEL
LIN {X 0,Y 472.772,Z 818.474,A -85,B 0,C 180,E1 16222.379,E2 16222.379} C_VEL
LIN {X 0,Y 476.374,Z 782.653,A -85,B 0,C 180,E1 16221.791,E2 16221.791} C_VEL
LIN {X 0,Y 494.946,Z 560.453,A -85,B 0,C 180,E1 16218.381,E2 16218.381} C_VEL
LIN {X 0,Y 495.804,Z 550.184,A -85,B 0,C 180,E1 16218.215,E2 16218.215} C_VEL
LIN {X 0,Y 490.833,Z 541.905,A -85,B 0,C 180,E1 16215.902,E2 16215.902} C_VEL
LIN {X 0,Y 486.516,Z 534.972,A -85,B 0,C 180,E1 16213.55,E2 16213.55} C_VEL
LIN {X 0,Y 483.616,Z 530.479,A -85,B 0,C 180,E1 16211.69,E2 16211.69} C_VEL
LIN {X 0,Y 481.166,Z 526.519,A -85,B 0,C 180,E1 16209.811,E2 16209.811} C_VEL
LIN {X 0,Y 478.311,Z 521.909,A -85,B 0,C 180,E1 16206.964,E2 16206.964} C_VEL
LIN {X 0,Y 475.887,Z 517.777,A -85,B 0,C 180,E1 16202.529,E2 16202.529} C_VEL
LIN {X 0,Y 475.759,Z 516.732,A -85,B 0,C 180,E1 16201.566,E2 16201.566} C_VEL
LIN {X 0,Y 475.797,Z 516.95,A -85,B 0,C 180,E1 16198.555,E2 16198.555} C_VEL
LIN {X 0,Y 477.477,Z 521.128,A -85,B 0,C 180,E1 16194.472,E2 16194.472} C_VEL
LIN {X 0,Y 478.723,Z 522.48,A -85,B 0,C 180,E1 16192.982,E2 16192.982} C_VEL
LIN {X 0,Y 482.182,Z 528.111,A -85,B 0,C 180,E1 16189.787,E2 16189.787} C_VEL
LIN {X 0,Y 485.1,Z 532.711,A -85,B 0,C 180,E1 16187.743,E2 16187.743} C_VEL
LIN {X 0,Y 488.208,Z 537.714,A -85,B 0,C 180,E1 16185.894,E2 16185.894} C_VEL
LIN {X 0,Y 493.937,Z 548.501,A -85,B 0,C 180,E1 16182.961,E2 16182.961} C_VEL
LIN {X 0,Y 495.89,Z 552.623,A -85,B 0,C 180,E1 16182.06,E2 16182.06} C_VEL
LIN {X 0,Y 477.436,Z 773.679,A -85,B 0,C 180,E1 16178.664,E2 16178.664} C_VEL
LIN {X 0,Y 473.134,Z 822.672,A -85,B 0,C 180,E1 16177.887,E2 16177.887} C_VEL
LIN {X 0,Y 468.839,Z 851.699,A -85,B 0,C 180,E1 16177.332,E2 16177.332} C_VEL
LIN {X 0,Y 464.413,Z 874.046,A -85,B 0,C 180,E1 16176.8,E2 16176.8} C_VEL
LIN {X 0,Y 459.548,Z 894.684,A -85,B 0,C 180,E1 16176.191,E2 16176.191} C_VEL
LIN {X 0,Y 453.732,Z 915.955,A -85,B 0,C 180,E1 16175.434,E2 16175.434} C_VEL
LIN {X 0,Y 445.898,Z 941.105,A -85,B 0,C 180,E1 16174.345,E2 16174.345} C_VEL
LIN {X 0,Y 436.959,Z 965.657,A -85,B 0,C 180,E1 16173.032,E2 16173.032} C_VEL
LIN {X 0,Y 429.45,Z 984.477,A -85,B 0,C 180,E1 16171.84,E2 16171.84} C_VEL
LIN {X 0,Y 421.542,Z 1002.691,A -85,B 0,C 180,E1 16170.515,E2 16170.515} C_VEL
LIN {X 0,Y 412.884,Z 1021.284,A -85,B 0,C 180,E1 16168.947,E2 16168.947} C_VEL
LIN {X 0,Y 402.088,Z 1043.019,A -85,B 0,C 180,E1 16166.8,E2 16166.8} C_VEL
LIN {X 0,Y 391.135,Z 1063.305,A -85,B 0,C 180,E1 16164.38,E2 16164.38} C_VEL
LIN {X 0,Y 382.247,Z 1079.115,A -85,B 0,C 180,E1 16162.181,E2 16162.181} C_VEL
LIN {X 0,Y 373.413,Z 1094.329,A -85,B 0,C 180,E1 16159.74,E2 16159.74} C_VEL
LIN {X 0,Y 363.224,Z 1111.579,A -85,B 0,C 180,E1 16156.511,E2 16156.511} C_VEL
LIN {X 0,Y 353.552,Z 1127.521,A -85,B 0,C 180,E1 16152.905,E2 16152.905} C_VEL
LIN {X 0,Y 346.234,Z 1139.763,A -85,B 0,C 180,E1 16149.658,E2 16149.658} C_VEL
LIN {X 0,Y 339.782,Z 1150.817,A -85,B 0,C 180,E1 16146.261,E2 16146.261} C_VEL
LIN {X 0,Y 333.127,Z 1163.03,A -85,B 0,C 180,E1 16141.849,E2 16141.849} C_VEL
LIN {X 0,Y 328.048,Z 1173.025,A -85,B 0,C 180,E1 16137.402,E2 16137.402} C_VEL
LIN {X 0,Y 324.769,Z 1180.479,A -85,B 0,C 180,E1 16133.44,E2 16133.44} C_VEL
LIN {X 0,Y 322.601,Z 1186.292,A -85,B 0,C 180,E1 16129.745,E2 16129.745} C_VEL
LIN {X 0,Y 321.145,Z 1191.329,A -85,B 0,C 180,E1 16125.829,E2 16125.829} C_VEL
LIN {X 0,Y 320.328,Z 1195.284,A -85,B 0,C 180,E1 16121.889,E2 16121.889} C_VEL
LIN {X 0,Y 320.019,Z 1198.405,A -85,B 0,C 180,E1 16117.54,E2 16117.54} C_VEL
LIN {X 0,Y 319.972,Z 1200.098,A -85,B 0,C 180,E1 16113.224,E2 16113.224} C_VEL
LIN {X 0,Y 319.975,Z 1200.407,A -85,B 0,C 180,E1 16109.105,E2 16109.105} C_VEL
LIN {X 0,Y 319.97,Z 1199.628,A -85,B 0,C 180,E1 16105.34,E2 16105.34} C_VEL
LIN {X 0,Y 320.048,Z 1197.809,A -85,B 0,C 180,E1 16101.557,E2 16101.557} C_VEL
LIN {X 0,Y 320.353,Z 1195.109,A -85,B 0,C 180,E1 16097.93,E2 16097.93} C_VEL
LIN {X 0,Y 321.164,Z 1191.234,A -85,B 0,C 180,E1 16094.1,E2 16094.1} C_VEL
LIN {X 0,Y 322.6,Z 1186.278,A -85,B 0,C 180,E1 16090.255,E2 16090.255} C_VEL
LIN {X 0,Y 324.767,Z 1180.462,A -85,B 0,C 180,E1 16086.561,E2 16086.561} C_VEL
LIN {X 0,Y 328.047,Z 1173,A -85,B 0,C 180,E1 16082.598,E2 16082.598} C_VEL
LIN {X 0,Y 333.405,Z 1162.455,A -85,B 0,C 180,E1 16077.94,E2 16077.94} C_VEL
LIN {X 0,Y 339.782,Z 1150.782,A -85,B 0,C 180,E1 16073.737,E2 16073.737} C_VEL
LIN {X 0,Y 346.23,Z 1139.723,A -85,B 0,C 180,E1 16070.341,E2 16070.341} C_VEL
LIN {X 0,Y 353.653,Z 1127.292,A -85,B 0,C 180,E1 16067.05,E2 16067.05} C_VEL
LIN {X 0,Y 363.411,Z 1111.162,A -85,B 0,C 180,E1 16063.419,E2 16063.419} C_VEL
LIN {X 0,Y 373.402,Z 1094.244,A -85,B 0,C 180,E1 16060.258,E2 16060.258} C_VEL
LIN {X 0,Y 382.235,Z 1079.019,A -85,B 0,C 180,E1 16057.817,E2 16057.817} C_VEL
LIN {X 0,Y 391.493,Z 1062.532,A -85,B 0,C 180,E1 16055.531,E2 16055.531} C_VEL
LIN {X 0,Y 402.986,Z 1041.047,A -85,B 0,C 180,E1 16053.006,E2 16053.006} C_VEL
LIN {X 0,Y 413.017,Z 1020.796,A -85,B 0,C 180,E1 16051.021,E2 16051.021} C_VEL
LIN {X 0,Y 421.523,Z 1002.495,A -85,B 0,C 180,E1 16049.48,E2 16049.48} C_VEL
LIN {X 0,Y 429.657,Z 983.724,A -85,B 0,C 180,E1 16048.119,E2 16048.119} C_VEL
LIN {X 0,Y 438.358,Z 961.793,A -85,B 0,C 180,E1 16046.75,E2 16046.75} C_VEL
LIN {X 0,Y 447.318,Z 936.268,A -85,B 0,C 180,E1 16045.441,E2 16045.441} C_VEL
LIN {X 0,Y 453.918,Z 914.875,A -85,B 0,C 180,E1 16044.533,E2 16044.533} C_VEL
LIN {X 0,Y 459.528,Z 894.259,A -85,B 0,C 180,E1 16043.803,E2 16043.803} C_VEL
LIN {X 0,Y 464.452,Z 873.271,A -85,B 0,C 180,E1 16043.186,E2 16043.186} C_VEL
LIN {X 0,Y 469.111,Z 849.519,A -85,B 0,C 180,E1 16042.628,E2 16042.628} C_VEL
LIN {X 0,Y 473.265,Z 820.009,A -85,B 0,C 180,E1 16042.075,E2 16042.075} C_VEL
LIN {X 0,Y 479.025,Z 752.353,A -85,B 0,C 180,E1 16041.013,E2 16041.013} C_VEL
